    RBT5_STANDARD_WELD_DATA : WORD ;
    RBT6_STANDARD_WELD_DATA : WORD ;
    RBT7_STANDARD_WELD_DATA : WORD ;
    RBT8_STANDARD_WELD_DATA : WORD ;
    RBT9_STANDARD_WELD_DATA : WORD ;
    RBT10_STANDARD_WELD_DATA : WORD ;
    RBT11_STANDARD_WELD_DATA : WORD ;
    RBT12_STANDARD_WELD_DATA : WORD ;
    RBT13_STANDARD_WELD_DATA : WORD ;
    RBT14_STANDARD_WELD_DATA : WORD ;
    RBT15_STANDARD_WELD_DATA : WORD ;
    RBT16_STANDARD_WELD_DATA : WORD ;
    RBT17_STANDARD_WELD_DATA : WORD ;
    RBT18_STANDARD_WELD_DATA : WORD ;
    RBT19_STANDARD_WELD_DATA : WORD ;
    RBT20_STANDARD_WELD_DATA : WORD ;
    RBT21_STANDARD_WELD_DATA : WORD ;
    RBT22_STANDARD_WELD_DATA : WORD ;
    RBT23_STANDARD_WELD_DAT : WORD ;
    RBT24_STANDARD_WELD_DAT : WORD ;
    CHK_WORD : WORD ;
    TEST_TEMP : ARRAY  [1 .. 40 ] OF BYTE ;
   END_STRUCT ;
   S705_BT_CODE_2117 : STRUCT
    STATION_MAIN : WORD ;
    DISTINCTION_LH_RH : WORD ;
    STAION_NUMBER : WORD ;
    BODY_TYPE_1ST : WORD ;
    BODY_TYPE_OPTION : WORD ;
    RBT1_STANDARD_WELD_DATA : WORD ;
    RBT2_STANDARD_WELD_DATA : WORD ;
    RBT3_STANDARD_WELD_DATA : WORD ;
    RBT4_STANDARD_WELD_DATA : WORD ;
    RBT5_STANDARD_WELD_DATA : WORD ;
    RBT6_STANDARD_WELD_DATA : WORD ;
    RBT7_STANDARD_WELD_DATA : WORD ;
    RBT8_STANDARD_WELD_DATA : WORD ;
    RBT9_STANDARD_WELD_DATA : WORD ;
    RBT10_STANDARD_WELD_DATA : WORD ;
    RBT11_STANDARD_WELD_DATA : WORD ;
    RBT12_STANDARD_WELD_DATA : WORD ;
    RBT13_STANDARD_WELD_DATA : WORD ;
    RBT14_STANDARD_WELD_DATA : WORD ;
    RBT15_STANDARD_WELD_DATA : WORD ;
    RBT16_STANDARD_WELD_DATA : WORD ;
    RBT17_STANDARD_WELD_DATA : WORD ;
    RBT18_STANDARD_WELD_DATA : WORD ;
    RBT19_STANDARD_WELD_DATA : WORD ;
    RBT20_STANDARD_WELD_DATA : WORD ;
    RBT21_STANDARD_WELD_DATA : WORD ;
    RBT22_STANDARD_WELD_DATA : WORD ;
    RBT23_STANDARD_WELD_DAT : WORD ;
    RBT24_STANDARD_WELD_DAT : WORD ;
    CHK_WORD : WORD ;
    TEST_TEMP : ARRAY  [1 .. 40 ] OF BYTE ;
   END_STRUCT ;
   S705_BT_CODE_2118 : STRUCT
    STATION_MAIN : WORD ;
    DISTINCTION_LH_RH : WORD ;
    STAION_NUMBER : WORD ;
    BODY_TYPE_1ST : WORD ;
    BODY_TYPE_OPTION : WORD ;
    RBT1_STANDARD_WELD_DATA : WORD ;
    RBT2_STANDARD_WELD_DATA : WORD ;
    RBT3_STANDARD_WELD_DATA : WORD ;
    RBT4_STANDARD_WELD_DATA : WORD ;
    RBT5_STANDARD_WELD_DATA : WORD ;
    RBT6_STANDARD_WELD_DATA : WORD ;
    RBT7_STANDARD_WELD_DATA : WORD ;
    RBT8_STANDARD_WELD_DATA : WORD ;
    RBT9_STANDARD_WELD_DATA : WORD ;
    RBT10_STANDARD_WELD_DATA : WORD ;
    RBT11_STANDARD_WELD_DATA : WORD ;
    RBT12_STANDARD_WELD_DATA : WORD ;
    RBT13_STANDARD_WELD_DATA : WORD ;
    RBT14_STANDARD_WELD_DATA : WORD ;
    RBT15_STANDARD_WELD_DATA : WORD ;
    RBT16_STANDARD_WELD_DATA : WORD ;
    RBT17_STANDARD_WELD_DATA : WORD ;
    RBT18_STANDARD_WELD_DATA : WORD ;
    RBT19_STANDARD_WELD_DATA : WORD ;
    RBT20_STANDARD_WELD_DATA : WORD ;
    RBT21_STANDARD_WELD_DATA : WORD ;
    RBT22_STANDARD_WELD_DATA : WORD ;
    RBT23_STANDARD_WELD_DAT : WORD ;
    RBT24_STANDARD_WELD_DAT : WORD ;
    CHK_WORD : WORD ;
    TEST_TEMP : ARRAY  [1 .. 40 ] OF BYTE ;
   END_STRUCT ;
   S705_BT_CODE_2119 : STRUCT
    STATION_MAIN : WORD ;
    DISTINCTION_LH_RH : WORD ;
    STAION_NUMBER : WORD ;
    BODY_TYPE_1ST : WORD ;
    BODY_TYPE_OPTION : WORD ;
    RBT1_STANDARD_WELD_DATA : WORD ;
    RBT2_STANDARD_WELD_DATA : WORD ;
    RBT3_STANDARD_WELD_DATA : WORD ;
    RBT4_STANDARD_WELD_DATA : WORD ;
    RBT5_STANDARD_WELD_DATA : WORD ;
    RBT6_STANDARD_WELD_DATA : WORD ;
    RBT7_STANDARD_WELD_DATA : WORD ;
    RBT8_STANDARD_WELD_DATA : WORD ;
    RBT9_STANDARD_WELD_DATA : WORD ;
    RBT10_STANDARD_WELD_DATA : WORD ;
    RBT11_STANDARD_WELD_DATA : WORD ;
    RBT12_STANDARD_WELD_DATA : WORD ;
    RBT13_STANDARD_WELD_DATA : WORD ;
    RBT14_STANDARD_WELD_DATA : WORD ;
    RBT15_STANDARD_WELD_DATA : WORD ;
    RBT16_STANDARD_WELD_DATA : WORD ;
    RBT17_STANDARD_WELD_DATA : WORD ;
    RBT18_STANDARD_WELD_DATA : WORD ;
    RBT19_STANDARD_WELD_DATA : WORD ;
    RBT20_STANDARD_WELD_DATA : WORD ;
    RBT21_STANDARD_WELD_DATA : WORD ;
    RBT22_STANDARD_WELD_DATA : WORD ;
    RBT23_STANDARD_WELD_DAT : WORD ;
    RBT24_STANDARD_WELD_DAT : WORD ;
    CHK_WORD : WORD ;
    TEST_TEMP : ARRAY  [1 .. 40 ] OF BYTE ;
   END_STRUCT ;
   S705_BT_CODE_2120 : STRUCT
    STATION_MAIN : WORD ;
    DISTINCTION_LH_RH : WORD ;
    STAION_NUMBER : WORD ;
    BODY_TYPE_1ST : WORD ;
    BODY_TYPE_OPTION : WORD ;
    RBT1_STANDARD_WELD_DATA : WORD ;
    RBT2_STANDARD_WELD_DATA : WORD ;
    RBT3_STANDARD_WELD_DATA : WORD ;
    RBT4_STANDARD_WELD_DATA : WORD ;
    RBT5_STANDARD_WELD_DATA : WORD ;
    RBT6_STANDARD_WELD_DATA : WORD ;
    RBT7_STANDARD_WELD_DATA : WORD ;
    RBT8_STANDARD_WELD_DATA : WORD ;
    RBT9_STANDARD_WELD_DATA : WORD ;
    RBT10_STANDARD_WELD_DATA : WORD ;
    RBT11_STANDARD_WELD_DATA : WORD ;
    RBT12_STANDARD_WELD_DATA : WORD ;
    RBT13_STANDARD_WELD_DATA : WORD ;
    RBT14_STANDARD_WELD_DATA : WORD ;
    RBT15_STANDARD_WELD_DATA : WORD ;
    RBT16_STANDARD_WELD_DATA : WORD ;
    RBT17_STANDARD_WELD_DATA : WORD ;
    RBT18_STANDARD_WELD_DATA : WORD ;
    RBT19_STANDARD_WELD_DATA : WORD ;
    RBT20_STANDARD_WELD_DATA : WORD ;
    RBT21_STANDARD_WELD_DATA : WORD ;
    RBT22_STANDARD_WELD_DATA : WORD ;
    RBT23_STANDARD_WELD_DAT : WORD ;
    RBT24_STANDARD_WELD_DAT : WORD ;
    CHK_WORD : WORD ;
    TEST_TEMP : ARRAY  [1 .. 40 ] OF BYTE ;
   END_STRUCT ;
   S706_BT_CODE_2101 : STRUCT
    STATION_MAIN : WORD ;
    DISTINCTION_LH_RH : WORD ;
    STAION_NUMBER : WORD ;
    BODY_TYPE_1ST : WORD ;
    BODY_TYPE_OPTION : WORD ;
    RBT1_STANDARD_WELD_DATA : WORD ;
    RBT2_STANDARD_WELD_DATA : WORD ;
    RBT3_STANDARD_WELD_DATA : WORD ;
    RBT4_STANDARD_WELD_DATA : WORD ;
    RBT5_STANDARD_WELD_DATA : WORD ;
    RBT6_STANDARD_WELD_DATA : WORD ;
    RBT7_STANDARD_WELD_DATA : WORD ;
    RBT8_STANDARD_WELD_DATA : WORD ;
    RBT9_STANDARD_WELD_DATA : WORD ;
    RBT10_STANDARD_WELD_DATA : WORD ;
    RBT11_STANDARD_WELD_DATA : WORD ;
    RBT12_STANDARD_WELD_DATA : WORD ;
    RBT13_STANDARD_WELD_DATA : WORD ;
    RBT14_STANDARD_WELD_DATA : WORD ;
    RBT15_STANDARD_WELD_DATA : WORD ;
    RBT16_STANDARD_WELD_DATA : WORD ;
    RBT17_STANDARD_WELD_DATA : WORD ;
    RBT18_STANDARD_WELD_DATA : WORD ;
    RBT19_STANDARD_WELD_DATA : WORD ;
    RBT20_STANDARD_WELD_DATA : WORD ;
    RBT21_STANDARD_WELD_DATA : WORD ;
    RBT22_STANDARD_WELD_DATA : WORD ;
    RBT23_STANDARD_WELD_DAT : WORD ;
    RBT24_STANDARD_WELD_DAT : WORD ;
    CHK_WORD : WORD ;
    TEST_TEMP : ARRAY  [1 .. 40 ] OF BYTE ;
   END_STRUCT ;
   S706_BT_CODE_2102 : STRUCT
    STATION_MAIN : WORD ;
    DISTINCTION_LH_RH : WORD ;
    STAION_NUMBER : WORD ;
    BODY_TYPE_1ST : WORD ;
    BODY_TYPE_OPTION : WORD ;
    RBT1_STANDARD_WELD_DATA : WORD ;
    RBT2_STANDARD_WELD_DATA : WORD ;
    RBT3_STANDARD_WELD_DATA : WORD ;
    RBT4_STANDARD_WELD_DATA : WORD ;
    RBT5_STANDARD_WELD_DATA : WORD ;
    RBT6_STANDARD_WELD_DATA : WORD ;
    RBT7_STANDARD_WELD_DATA : WORD ;
    RBT8_STANDARD_WELD_DATA : WORD ;
    RBT9_STANDARD_WELD_DATA : WORD ;
    RBT10_STANDARD_WELD_DATA : WORD ;
    RBT11_STANDARD_WELD_DATA : WORD ;
    RBT12_STANDARD_WELD_DATA : WORD ;
    RBT13_STANDARD_WELD_DATA : WORD ;
    RBT14_STANDARD_WELD_DATA : WORD ;
    RBT15_STANDARD_WELD_DATA : WORD ;
    RBT16_STANDARD_WELD_DATA : WORD ;
    RBT17_STANDARD_WELD_DATA : WORD ;
    RBT18_STANDARD_WELD_DATA : WORD ;
    RBT19_STANDARD_WELD_DATA : WORD ;
    RBT20_STANDARD_WELD_DATA : WORD ;
    RBT21_STANDARD_WELD_DATA : WORD ;
    RBT22_STANDARD_WELD_DATA : WORD ;
    RBT23_STANDARD_WELD_DAT : WORD ;
    RBT24_STANDARD_WELD_DAT : WORD ;
    CHK_WORD : WORD ;
    TEST_TEMP : ARRAY  [1 .. 40 ] OF BYTE ;
   END_STRUCT ;
   S706_BT_CODE_2103 : STRUCT
    STATION_MAIN : WORD ;
    DISTINCTION_LH_RH : WORD ;
    STAION_NUMBER : WORD ;
    BODY_TYPE_1ST : WORD ;
    BODY_TYPE_OPTION : WORD ;
    RBT1_STANDARD_WELD_DATA : WORD ;
    RBT2_STANDARD_WELD_DATA : WORD ;
    RBT3_STANDARD_WELD_DATA : WORD ;
    RBT4_STANDARD_WELD_DATA : WORD ;
    RBT5_STANDARD_WELD_DATA : WORD ;
    RBT6_STANDARD_WELD_DATA : WORD ;
    RBT7_STANDARD_WELD_DATA : WORD ;
    RBT8_STANDARD_WELD_DATA : WORD ;
    RBT9_STANDARD_WELD_DATA : WORD ;
    RBT10_STANDARD_WELD_DATA : WORD ;
    RBT11_STANDARD_WELD_DATA : WORD ;
    RBT12_STANDARD_WELD_DATA : WORD ;
    RBT13_STANDARD_WELD_DATA : WORD ;
    RBT14_STANDARD_WELD_DATA : WORD ;
    RBT15_STANDARD_WELD_DATA : WORD ;
    RBT16_STANDARD_WELD_DATA : WORD ;
    RBT17_STANDARD_WELD_DATA : WORD ;
    RBT18_STANDARD_WELD_DATA : WORD ;
    RBT19_STANDARD_WELD_DATA : WORD ;
    RBT20_STANDARD_WELD_DATA : WORD ;
    RBT21_STANDARD_WELD_DATA : WORD ;
    RBT22_STANDARD_WELD_DATA : WORD ;
    RBT23_STANDARD_WELD_DAT : WORD ;
    RBT24_STANDARD_WELD_DAT : WORD ;
    CHK_WORD : WORD ;
    TEST_TEMP : ARRAY  [1 .. 40 ] OF BYTE ;
   END_STRUCT ;
   S706_BT_CODE_2104 : STRUCT
    STATION_MAIN : WORD ;
    DISTINCTION_LH_RH : WORD ;
    STAION_NUMBER : WORD ;
    BODY_TYPE_1ST : WORD ;
    BODY_TYPE_OPTION : WORD ;
    RBT1_STANDARD_WELD_DATA : WORD ;
    RBT2_STANDARD_WELD_DATA : WORD ;
    RBT3_STANDARD_WELD_DATA : WORD ;
    RBT4_STANDARD_WELD_DATA : WORD ;
    RBT5_STANDARD_WELD_DATA : WORD ;
    RBT6_STANDARD_WELD_DATA : WORD ;
    RBT7_STANDARD_WELD_DATA : WORD ;
    RBT8_STANDARD_WELD_DATA : WORD ;
    RBT9_STANDARD_WELD_DATA : WORD ;
    RBT10_STANDARD_WELD_DATA : WORD ;
    RBT11_STANDARD_WELD_DATA : WORD ;
    RBT12_STANDARD_WELD_DATA : WORD ;
    RBT13_STANDARD_WELD_DATA : WORD ;
    RBT14_STANDARD_WELD_DATA : WORD ;
    RBT15_STANDARD_WELD_DATA : WORD ;
    RBT16_STANDARD_WELD_DATA : WORD ;
    RBT17_STANDARD_WELD_DATA : WORD ;
    RBT18_STANDARD_WELD_DATA : WORD ;
    RBT19_STANDARD_WELD_DATA : WORD ;
    RBT20_STANDARD_WELD_DATA : WORD ;
    RBT21_STANDARD_WELD_DATA : WORD ;
    RBT22_STANDARD_WELD_DATA : WORD ;
    RBT23_STANDARD_WELD_DAT : WORD ;
    RBT24_STANDARD_WELD_DAT : WORD ;
    CHK_WORD : WORD ;
    TEST_TEMP : ARRAY  [1 .. 40 ] OF BYTE ;
   END_STRUCT ;
   S706_BT_CODE_2105 : STRUCT
    STATION_MAIN : WORD ;
    DISTINCTION_LH_RH : WORD ;
    STAION_NUMBER : WORD ;
    BODY_TYPE_1ST : WORD ;
    BODY_TYPE_OPTION : WORD ;
    RBT1_STANDARD_WELD_DATA : WORD ;
    RBT2_STANDARD_WELD_DATA : WORD ;
    RBT3_STANDARD_WELD_DATA : WORD ;
    RBT4_STANDARD_WELD_DATA : WORD ;
    RBT5_STANDARD_WELD_DATA : WORD ;
    RBT6_STANDARD_WELD_DATA : WORD ;
    RBT7_STANDARD_WELD_DATA : WORD ;
    RBT8_STANDARD_WELD_DATA : WORD ;
    RBT9_STANDARD_WELD_DATA : WORD ;
    RBT10_STANDARD_WELD_DATA : WORD ;
    RBT11_STANDARD_WELD_DATA : WORD ;
    RBT12_STANDARD_WELD_DATA : WORD ;
    RBT13_STANDARD_WELD_DATA : WORD ;
    RBT14_STANDARD_WELD_DATA : WORD ;
    RBT15_STANDARD_WELD_DATA : WORD ;
    RBT16_STANDARD_WELD_DATA : WORD ;
    RBT17_STANDARD_WELD_DATA : WORD ;
    RBT18_STANDARD_WELD_DATA : WORD ;
    RBT19_STANDARD_WELD_DATA : WORD ;
    RBT20_STANDARD_WELD_DATA : WORD ;
    RBT21_STANDARD_WELD_DATA : WORD ;
    RBT22_STANDARD_WELD_DATA : WORD ;
    RBT23_STANDARD_WELD_DAT : WORD ;
    RBT24_STANDARD_WELD_DAT : WORD ;
    CHK_WORD : WORD ;
    TEST_TEMP : ARRAY  [1 .. 40 ] OF BYTE ;
   END_STRUCT ;
   S706_BT_CODE_2106 : STRUCT
    STATION_MAIN : WORD ;
    DISTINCTION_LH_RH : WORD ;
    STAION_NUMBER : WORD ;
    BODY_TYPE_1ST : WORD ;
    BODY_TYPE_OPTION : WORD ;
    RBT1_STANDARD_WELD_DATA : WORD ;
    RBT2_STANDARD_WELD_DATA : WORD ;
    RBT3_STANDARD_WELD_DATA : WORD ;
    RBT4_STANDARD_WELD_DATA : WORD ;
    RBT5_STANDARD_WELD_DATA : WORD ;
    RBT6_STANDARD_WELD_DATA : WORD ;
    RBT7_STANDARD_WELD_DATA : WORD ;
    RBT8_STANDARD_WELD_DATA : WORD ;
    RBT9_STANDARD_WELD_DATA : WORD ;
    RBT10_STANDARD_WELD_DATA : WORD ;
    RBT11_STANDARD_WELD_DATA : WORD ;
    RBT12_STANDARD_WELD_DATA : WORD ;
    RBT13_STANDARD_WELD_DATA : WORD ;
    RBT14_STANDARD_WELD_DATA : WORD ;
    RBT15_STANDARD_WELD_DATA : WORD ;
    RBT16_STANDARD_WELD_DATA : WORD ;
    RBT17_STANDARD_WELD_DATA : WORD ;
    RBT18_STANDARD_WELD_DATA : WORD ;
    RBT19_STANDARD_WELD_DATA : WORD ;
    RBT20_STANDARD_WELD_DATA : WORD ;
    RBT21_STANDARD_WELD_DATA : WORD ;
    RBT22_STANDARD_WELD_DATA : WORD ;
    RBT23_STANDARD_WELD_DAT : WORD ;
    RBT24_STANDARD_WELD_DAT : WORD ;
    CHK_WORD : WORD ;
    TEST_TEMP : ARRAY  [1 .. 40 ] OF BYTE ;
   END_STRUCT ;
   S706_BT_CODE_2107 : STRUCT
    STATION_MAIN : WORD ;
    DISTINCTION_LH_RH : WORD ;
    STAION_NUMBER : WORD ;
    BODY_TYPE_1ST : WORD ;
    BODY_TYPE_OPTION : WORD ;
    RBT1_STANDARD_WELD_DATA : WORD ;
    RBT2_STANDARD_WELD_DATA : WORD ;
    RBT3_STANDARD_WELD_DATA : WORD ;
    RBT4_STANDARD_WELD_DATA : WORD ;
    RBT5_STANDARD_WELD_DATA : WORD ;
    RBT6_STANDARD_WELD_DATA : WORD ;
    RBT7_STANDARD_WELD_DATA : WORD ;
    RBT8_STANDARD_WELD_DATA : WORD ;
    RBT9_STANDARD_WELD_DATA : WORD ;
    RBT10_STANDARD_WELD_DATA : WORD ;
    RBT11_STANDARD_WELD_DATA : WORD ;
    RBT12_STANDARD_WELD_DATA : WORD ;
    RBT13_STANDARD_WELD_DATA : WORD ;
    RBT14_STANDARD_WELD_DATA : WORD ;
    RBT15_STANDARD_WELD_DATA : WORD ;
    RBT16_STANDARD_WELD_DATA : WORD ;
    RBT17_STANDARD_WELD_DATA : WORD ;
    RBT18_STANDARD_WELD_DATA : WORD ;
    RBT19_STANDARD_WELD_DATA : WORD ;
    RBT20_STANDARD_WELD_DATA : WORD ;
    RBT21_STANDARD_WELD_DATA : WORD ;
    RBT22_STANDARD_WELD_DATA : WORD ;
    RBT23_STANDARD_WELD_DAT : WORD ;
    RBT24_STANDARD_WELD_DAT : WORD ;
    CHK_WORD : WORD ;
    TEST_TEMP : ARRAY  [1 .. 40 ] OF BYTE ;
   END_STRUCT ;
   S706_BT_CODE_2108 : STRUCT
    STATION_MAIN : WORD ;
    DISTINCTION_LH_RH : WORD ;
    STAION_NUMBER : WORD ;
    BODY_TYPE_1ST : WORD ;
    BODY_TYPE_OPTION : WORD ;
    RBT1_STANDARD_WELD_DATA : WORD ;
    RBT2_STANDARD_WELD_DATA : WORD ;
    RBT3_STANDARD_WELD_DATA : WORD ;
    RBT4_STANDARD_WELD_DATA : WORD ;
    RBT5_STANDARD_WELD_DATA : WORD ;
    RBT6_STANDARD_WELD_DATA : WORD ;
    RBT7_STANDARD_WELD_DATA : WORD ;
    RBT8_STANDARD_WELD_DATA : WORD ;
    RBT9_STANDARD_WELD_DATA : WORD ;
    RBT10_STANDARD_WELD_DATA : WORD ;
    RBT11_STANDARD_WELD_DATA : WORD ;
    RBT12_STANDARD_WELD_DATA : WORD ;
    RBT13_STANDARD_WELD_DATA : WORD ;
    RBT14_STANDARD_WELD_DATA : WORD ;
    RBT15_STANDARD_WELD_DATA : WORD ;
    RBT16_STANDARD_WELD_DATA : WORD ;
    RBT17_STANDARD_WELD_DATA : WORD ;
    RBT18_STANDARD_WELD_DATA : WORD ;
    RBT19_STANDARD_WELD_DATA : WORD ;
    RBT20_STANDARD_WELD_DATA : WORD ;
    RBT21_STANDARD_WELD_DATA : WORD ;
    RBT22_STANDARD_WELD_DATA : WORD ;
    RBT23_STANDARD_WELD_DAT : WORD ;
    RBT24_STANDARD_WELD_DAT : WORD ;
    CHK_WORD : WORD ;
    TEST_TEMP : ARRAY  [1 .. 40 ] OF BYTE ;
   END_STRUCT ;
   S706_BT_CODE_2109 : STRUCT
    STATION_MAIN : WORD ;
    DISTINCTION_LH_RH : WORD ;
    STAION_NUMBER : WORD ;
    BODY_TYPE_1ST : WORD ;
    BODY_TYPE_OPTION : WORD ;
    RBT1_STANDARD_WELD_DATA : WORD ;
    RBT2_STANDARD_WELD_DATA : WORD ;
    RBT3_STANDARD_WELD_DATA : WORD ;
    RBT4_STANDARD_WELD_DATA : WORD ;
    RBT5_STANDARD_WELD_DATA : WORD ;
    RBT6_STANDARD_WELD_DATA : WORD ;
    RBT7_STANDARD_WELD_DATA : WORD ;
    RBT8_STANDARD_WELD_DATA : WORD ;
    RBT9_STANDARD_WELD_DATA : WORD ;
    RBT10_STANDARD_WELD_DATA : WORD ;
    RBT11_STANDARD_WELD_DATA : WORD ;
    RBT12_STANDARD_WELD_DATA : WORD ;
    RBT13_STANDARD_WELD_DATA : WORD ;
    RBT14_STANDARD_WELD_DATA : WORD ;
    RBT15_STANDARD_WELD_DATA : WORD ;
    RBT16_STANDARD_WELD_DATA : WORD ;
    RBT17_STANDARD_WELD_DATA : WORD ;
    RBT18_STANDARD_WELD_DATA : WORD ;
    RBT19_STANDARD_WELD_DATA : WORD ;
    RBT20_STANDARD_WELD_DATA : WORD ;
    RBT21_STANDARD_WELD_DATA : WORD ;
    RBT22_STANDARD_WELD_DATA : WORD ;
    RBT23_STANDARD_WELD_DAT : WORD ;
    RBT24_STANDARD_WELD_DAT : WORD ;
    CHK_WORD : WORD ;
    TEST_TEMP : ARRAY  [1 .. 40 ] OF BYTE ;
   END_STRUCT ;
   S706_BT_CODE_2110 : STRUCT
    STATION_MAIN : WORD ;
    DISTINCTION_LH_RH : WORD ;
    STAION_NUMBER : WORD ;
    BODY_TYPE_1ST : WORD ;
    BODY_TYPE_OPTION : WORD ;
    RBT1_STANDARD_WELD_DATA : WORD ;
    RBT2_STANDARD_WELD_DATA : WORD ;
    RBT3_STANDARD_WELD_DATA : WORD ;
    RBT4_STANDARD_WELD_DATA : WORD ;
    RBT5_STANDARD_WELD_DATA : WORD ;
    RBT6_STANDARD_WELD_DATA : WORD ;
    RBT7_STANDARD_WELD_DATA : WORD ;
    RBT8_STANDARD_WELD_DATA : WORD ;
    RBT9_STANDARD_WELD_DATA : WORD ;
    RBT10_STANDARD_WELD_DATA : WORD ;
    RBT11_STANDARD_WELD_DATA : WORD ;
    RBT12_STANDARD_WELD_DATA : WORD ;
    RBT13_STANDARD_WELD_DATA : WORD ;
    RBT14_STANDARD_WELD_DATA : WORD ;
    RBT15_STANDARD_WELD_DATA : WORD ;
    RBT16_STANDARD_WELD_DATA : WORD ;
    RBT17_STANDARD_WELD_DATA : WORD ;
    RBT18_STANDARD_WELD_DATA : WORD ;
    RBT19_STANDARD_WELD_DATA : WORD ;
    RBT20_STANDARD_WELD_DATA : WORD ;
    RBT21_STANDARD_WELD_DATA : WORD ;
    RBT22_STANDARD_WELD_DATA : WORD ;
    RBT23_STANDARD_WELD_DAT : WORD ;
    RBT24_STANDARD_WELD_DAT : WORD ;
    CHK_WORD : WORD ;
    TEST_TEMP : ARRAY  [1 .. 40 ] OF BYTE ;
   END_STRUCT ;
   S706_BT_CODE_2111 : STRUCT
    STATION_MAIN : WORD ;
    DISTINCTION_LH_RH : WORD ;
    STAION_NUMBER : WORD ;
    BODY_TYPE_1ST : WORD ;
    BODY_TYPE_OPTION : WORD ;
    RBT1_STANDARD_WELD_DATA : WORD ;
    RBT2_STANDARD_WELD_DATA : WORD ;
    RBT3_STANDARD_WELD_DATA : WORD ;
    RBT4_STANDARD_WELD_DATA : WORD ;
    RBT5_STANDARD_WELD_DATA : WORD ;
    RBT6_STANDARD_WELD_DATA : WORD ;
    RBT7_STANDARD_WELD_DATA : WORD ;
    RBT8_STANDARD_WELD_DATA : WORD ;
    RBT9_STANDARD_WELD_DATA : WORD ;
    RBT10_STANDARD_WELD_DATA : WORD ;
    RBT11_STANDARD_WELD_DATA : WORD ;
    RBT12_STANDARD_WELD_DATA : WORD ;
    RBT13_STANDARD_WELD_DATA : WORD ;
    RBT14_STANDARD_WELD_DATA : WORD ;
    RBT15_STANDARD_WELD_DATA : WORD ;
    RBT16_STANDARD_WELD_DATA : WORD ;
    RBT17_STANDARD_WELD_DATA : WORD ;
    RBT18_STANDARD_WELD_DATA : WORD ;
    RBT19_STANDARD_WELD_DATA : WORD ;
    RBT20_STANDARD_WELD_DATA : WORD ;
    RBT21_STANDARD_WELD_DATA : WORD ;
    RBT22_STANDARD_WELD_DATA : WORD ;
    RBT23_STANDARD_WELD_DAT : WORD ;
    RBT24_STANDARD_WELD_DAT : WORD ;
    CHK_WORD : WORD ;
    TEST_TEMP : ARRAY  [1 .. 40 ] OF BYTE ;
   END_STRUCT ;
   S706_BT_CODE_2112 : STRUCT
    STATION_MAIN : WORD ;
    DISTINCTION_LH_RH : WORD ;
    STAION_NUMBER : WORD ;
    BODY_TYPE_1ST : WORD ;
    BODY_TYPE_OPTION : WORD ;
    RBT1_STANDARD_WELD_DATA : WORD ;
    RBT2_STANDARD_WELD_DATA : WORD ;
    RBT3_STANDARD_WELD_DATA : WORD ;
    RBT4_STANDARD_WELD_DATA : WORD ;
    RBT5_STANDARD_WELD_DATA : WORD ;
    RBT6_STANDARD_WELD_DATA : WORD ;
    RBT7_STANDARD_WELD_DATA : WORD ;
    RBT8_STANDARD_WELD_DATA : WORD ;
    RBT9_STANDARD_WELD_DATA : WORD ;
    RBT10_STANDARD_WELD_DATA : WORD ;
    RBT11_STANDARD_WELD_DATA : WORD ;
    RBT12_STANDARD_WELD_DATA : WORD ;
    RBT13_STANDARD_WELD_DATA : WORD ;
    RBT14_STANDARD_WELD_DATA : WORD ;
    RBT15_STANDARD_WELD_DATA : WORD ;
    RBT16_STANDARD_WELD_DATA : WORD ;
    RBT17_STANDARD_WELD_DATA : WORD ;
    RBT18_STANDARD_WELD_DATA : WORD ;
    RBT19_STANDARD_WELD_DATA : WORD ;
    RBT20_STANDARD_WELD_DATA : WORD ;
    RBT21_STANDARD_WELD_DATA : WORD ;
    RBT22_STANDARD_WELD_DATA : WORD ;
    RBT23_STANDARD_WELD_DAT : WORD ;
    RBT24_STANDARD_WELD_DAT : WORD ;
    CHK_WORD : WORD ;
    TEST_TEMP : ARRAY  [1 .. 40 ] OF BYTE ;
   END_STRUCT ;
   S706_BT_CODE_2113 : STRUCT
    STATION_MAIN : WORD ;
    DISTINCTION_LH_RH : WORD ;
    STAION_NUMBER : WORD ;
    BODY_TYPE_1ST : WORD ;
    BODY_TYPE_OPTION : WORD ;
    RBT1_STANDARD_WELD_DATA : WORD ;
    RBT2_STANDARD_WELD_DATA : WORD ;
    RBT3_STANDARD_WELD_DATA : WORD ;
    RBT4_STANDARD_WELD_DATA : WORD ;
    RBT5_STANDARD_WELD_DATA : WORD ;
    RBT6_STANDARD_WELD_DATA : WORD ;
    RBT7_STANDARD_WELD_DATA : WORD ;
    RBT8_STANDARD_WELD_DATA : WORD ;
    RBT9_STANDARD_WELD_DATA : WORD ;
    RBT10_STANDARD_WELD_DATA : WORD ;
    RBT11_STANDARD_WELD_DATA : WORD ;
    RBT12_STANDARD_WELD_DATA : WORD ;
    RBT13_STANDARD_WELD_DATA : WORD ;
    RBT14_STANDARD_WELD_DATA : WORD ;
    RBT15_STANDARD_WELD_DATA : WORD ;
    RBT16_STANDARD_WELD_DATA : WORD ;
    RBT17_STANDARD_WELD_DATA : WORD ;
    RBT18_STANDARD_WELD_DATA : WORD ;
    RBT19_STANDARD_WELD_DATA : WORD ;
    RBT20_STANDARD_WELD_DATA : WORD ;
    RBT21_STANDARD_WELD_DATA : WORD ;
    RBT22_STANDARD_WELD_DATA : WORD ;
    RBT23_STANDARD_WELD_DAT : WORD ;
    RBT24_STANDARD_WELD_DAT : WORD ;
    CHK_WORD : WORD ;
    TEST_TEMP : ARRAY  [1 .. 40 ] OF BYTE ;
   END_STRUCT ;
   S706_BT_CODE_2114 : STRUCT
    STATION_MAIN : WORD ;
    DISTINCTION_LH_RH : WORD ;
    STAION_NUMBER : WORD ;
    BODY_TYPE_1ST : WORD ;
    BODY_TYPE_OPTION : WORD ;
    RBT1_STANDARD_WELD_DATA : WORD ;
    RBT2_STANDARD_WELD_DATA : WORD ;
    RBT3_STANDARD_WELD_DATA : WORD ;
    RBT4_STANDARD_WELD_DATA : WORD ;
    RBT5_STANDARD_WELD_DATA : WORD ;
    RBT6_STANDARD_WELD_DATA : WORD ;
    RBT7_STANDARD_WELD_DATA : WORD ;
    RBT8_STANDARD_WELD_DATA : WORD ;
    RBT9_STANDARD_WELD_DATA : WORD ;
    RBT10_STANDARD_WELD_DATA : WORD ;
    RBT11_STANDARD_WELD_DATA : WORD ;
    RBT12_STANDARD_WELD_DATA : WORD ;
    RBT13_STANDARD_WELD_DATA : WORD ;
    RBT14_STANDARD_WELD_DATA : WORD ;
    RBT15_STANDARD_WELD_DATA : WORD ;
    RBT16_STANDARD_WELD_DATA : WORD ;
    RBT17_STANDARD_WELD_DATA : WORD ;
    RBT18_STANDARD_WELD_DATA : WORD ;
    RBT19_STANDARD_WELD_DATA : WORD ;
    RBT20_STANDARD_WELD_DATA : WORD ;
    RBT21_STANDARD_WELD_DATA : WORD ;
    RBT22_STANDARD_WELD_DATA : WORD ;
    RBT23_STANDARD_WELD_DAT : WORD ;
    RBT24_STANDARD_WELD_DAT : WORD ;
    CHK_WORD : WORD ;
    TEST_TEMP : ARRAY  [1 .. 40 ] OF BYTE ;
   END_STRUCT ;
   S706_BT_CODE_2115 : STRUCT
    STATION_MAIN : WORD ;
    DISTINCTION_LH_RH : WORD ;
    STAION_NUMBER : WORD ;
    BODY_TYPE_1ST : WORD ;
    BODY_TYPE_OPTION : WORD ;
    RBT1_STANDARD_WELD_DATA : WORD ;
    RBT2_STANDARD_WELD_DATA : WORD ;
    RBT3_STANDARD_WELD_DATA : WORD ;
    RBT4_STANDARD_WELD_DATA : WORD ;
    RBT5_STANDARD_WELD_DATA : WORD ;
    RBT6_STANDARD_WELD_DATA : WORD ;
    RBT7_STANDARD_WELD_DATA : WORD ;
    RBT8_STANDARD_WELD_DATA : WORD ;
    RBT9_STANDARD_WELD_DATA : WORD ;
    RBT10_STANDARD_WELD_DATA : WORD ;
    RBT11_STANDARD_WELD_DATA : WORD ;
    RBT12_STANDARD_WELD_DATA : WORD ;
    RBT13_STANDARD_WELD_DATA : WORD ;
    RBT14_STANDARD_WELD_DATA : WORD ;
    RBT15_STANDARD_WELD_DATA : WORD ;
    RBT16_STANDARD_WELD_DATA : WORD ;
    RBT17_STANDARD_WELD_DATA : WORD ;
    RBT18_STANDARD_WELD_DATA : WORD ;
    RBT19_STANDARD_WELD_DATA : WORD ;
    RBT20_STANDARD_WELD_DATA : WORD ;
    RBT21_STANDARD_WELD_DATA : WORD ;
    RBT22_STANDARD_WELD_DATA : WORD ;
    RBT23_STANDARD_WELD_DAT : WORD ;
    RBT24_STANDARD_WELD_DAT : WORD ;
    CHK_WORD : WORD ;
    TEST_TEMP : ARRAY  [1 .. 40 ] OF BYTE ;
   END_STRUCT ;
   S706_BT_CODE_2116 : STRUCT
    STATION_MAIN : WORD ;
    DISTINCTION_LH_RH : WORD ;
    STAION_NUMBER : WORD ;
    BODY_TYPE_1ST : WORD ;
    BODY_TYPE_OPTION : WORD ;
    RBT1_STANDARD_WELD_DATA : WORD ;
    RBT2_STANDARD_WELD_DATA : WORD ;
    RBT3_STANDARD_WELD_DATA : WORD ;
    RBT4_STANDARD_WELD_DATA : WORD ;
    RBT5_STANDARD_WELD_DATA : WORD ;
    RBT6_STANDARD_WELD_DATA : WORD ;
    RBT7_STANDARD_WELD_DATA : WORD ;
    RBT8_STANDARD_WELD_DATA : WORD ;
    RBT9_STANDARD_WELD_DATA : WORD ;
    RBT10_STANDARD_WELD_DATA : WORD ;
    RBT11_STANDARD_WELD_DATA : WORD ;
    RBT12_STANDARD_WELD_DATA : WORD ;
    RBT13_STANDARD_WELD_DATA : WORD ;
    RBT14_STANDARD_WELD_DATA : WORD ;
    RBT15_STANDARD_WELD_DATA : WORD ;
    RBT16_STANDARD_WELD_DATA : WORD ;
    RBT17_STANDARD_WELD_DATA : WORD ;
    RBT18_STANDARD_WELD_DATA : WORD ;
    RBT19_STANDARD_WELD_DATA : WORD ;
    RBT20_STANDARD_WELD_DATA : WORD ;
    RBT21_STANDARD_WELD_DATA : WORD ;
    RBT22_STANDARD_WELD_DATA : WORD ;
    RBT23_STANDARD_WELD_DAT : WORD ;
    RBT24_STANDARD_WELD_DAT : WORD ;
    CHK_WORD : WORD ;
    TEST_TEMP : ARRAY  [1 .. 40 ] OF BYTE ;
   END_STRUCT ;
   S706_BT_CODE_2117 : STRUCT
    STATION_MAIN : WORD ;
    DISTINCTION_LH_RH : WORD ;
    STAION_NUMBER : WORD ;
    BODY_TYPE_1ST : WORD ;
    BODY_TYPE_OPTION : WORD ;
    RBT1_STANDARD_WELD_DATA : WORD ;
    RBT2_STANDARD_WELD_DATA : WORD ;
    RBT3_STANDARD_WELD_DATA : WORD ;
    RBT4_STANDARD_WELD_DATA : WORD ;
    RBT5_STANDARD_WELD_DATA : WORD ;
    RBT6_STANDARD_WELD_DATA : WORD ;
    RBT7_STANDARD_WELD_DATA : WORD ;
    RBT8_STANDARD_WELD_DATA : WORD ;
    RBT9_STANDARD_WELD_DATA : WORD ;
    RBT10_STANDARD_WELD_DATA : WORD ;
    RBT11_STANDARD_WELD_DATA : WORD ;
    RBT12_STANDARD_WELD_DATA : WORD ;
    RBT13_STANDARD_WELD_DATA : WORD ;
    RBT14_STANDARD_WELD_DATA : WORD ;
    RBT15_STANDARD_WELD_DATA : WORD ;
    RBT16_STANDARD_WELD_DATA : WORD ;
    RBT17_STANDARD_WELD_DATA : WORD ;
    RBT18_STANDARD_WELD_DATA : WORD ;
    RBT19_STANDARD_WELD_DATA : WORD ;
    RBT20_STANDARD_WELD_DATA : WORD ;
    RBT21_STANDARD_WELD_DATA : WORD ;
    RBT22_STANDARD_WELD_DATA : WORD ;
    RBT23_STANDARD_WELD_DAT : WORD ;
    RBT24_STANDARD_WELD_DAT : WORD ;
    CHK_WORD : WORD ;
    TEST_TEMP : ARRAY  [1 .. 40 ] OF BYTE ;
   END_STRUCT ;
   S706_BT_CODE_2118 : STRUCT
    STATION_MAIN : WORD ;
    DISTINCTION_LH_RH : WORD ;
    STAION_NUMBER : WORD ;
    BODY_TYPE_1ST : WORD ;
    BODY_TYPE_OPTION : WORD ;
    RBT1_STANDARD_WELD_DATA : WORD ;
    RBT2_STANDARD_WELD_DATA : WORD ;
    RBT3_STANDARD_WELD_DATA : WORD ;
    RBT4_STANDARD_WELD_DATA : WORD ;
    RBT5_STANDARD_WELD_DATA : WORD ;
    RBT6_STANDARD_WELD_DATA : WORD ;
    RBT7_STANDARD_WELD_DATA : WORD ;
    RBT8_STANDARD_WELD_DATA : WORD ;
    RBT9_STANDARD_WELD_DATA : WORD ;
    RBT10_STANDARD_WELD_DATA : WORD ;
    RBT11_STANDARD_WELD_DATA : WORD ;
    RBT12_STANDARD_WELD_DATA : WORD ;
    RBT13_STANDARD_WELD_DATA : WORD ;
    RBT14_STANDARD_WELD_DATA : WORD ;
    RBT15_STANDARD_WELD_DATA : WORD ;
    RBT16_STANDARD_WELD_DATA : WORD ;
    RBT17_STANDARD_WELD_DATA : WORD ;
    RBT18_STANDARD_WELD_DATA : WORD ;
    RBT19_STANDARD_WELD_DATA : WORD ;
    RBT20_STANDARD_WELD_DATA : WORD ;
    RBT21_STANDARD_WELD_DATA : WORD ;
    RBT22_STANDARD_WELD_DATA : WORD ;
    RBT23_STANDARD_WELD_DAT : WORD ;
    RBT24_STANDARD_WELD_DAT : WORD ;
    CHK_WORD : WORD ;
    TEST_TEMP : ARRAY  [1 .. 40 ] OF BYTE ;
   END_STRUCT ;
   S706_BT_CODE_2119 : STRUCT
    STATION_MAIN : WORD ;
    DISTINCTION_LH_RH : WORD ;
    STAION_NUMBER : WORD ;
    BODY_TYPE_1ST : WORD ;
    BODY_TYPE_OPTION : WORD ;
    RBT1_STANDARD_WELD_DATA : WORD ;
    RBT2_STANDARD_WELD_DATA : WORD ;
    RBT3_STANDARD_WELD_DATA : WORD ;
    RBT4_STANDARD_WELD_DATA : WORD ;
    RBT5_STANDARD_WELD_DATA : WORD ;
    RBT6_STANDARD_WELD_DATA : WORD ;
    RBT7_STANDARD_WELD_DATA : WORD ;
    RBT8_STANDARD_WELD_DATA : WORD ;
    RBT9_STANDARD_WELD_DATA : WORD ;
    RBT10_STANDARD_WELD_DATA : WORD ;
    RBT11_STANDARD_WELD_DATA : WORD ;
    RBT12_STANDARD_WELD_DATA : WORD ;
    RBT13_STANDARD_WELD_DATA : WORD ;
    RBT14_STANDARD_WELD_DATA : WORD ;
    RBT15_STANDARD_WELD_DATA : WORD ;
    RBT16_STANDARD_WELD_DATA : WORD ;
    RBT17_STANDARD_WELD_DATA : WORD ;
    RBT18_STANDARD_WELD_DATA : WORD ;
    RBT19_STANDARD_WELD_DATA : WORD ;
    RBT20_STANDARD_WELD_DATA : WORD ;
    RBT21_STANDARD_WELD_DATA : WORD ;
    RBT22_STANDARD_WELD_DATA : WORD ;
    RBT23_STANDARD_WELD_DAT : WORD ;
    RBT24_STANDARD_WELD_DAT : WORD ;
    CHK_WORD : WORD ;
    TEST_TEMP : ARRAY  [1 .. 40 ] OF BYTE ;
   END_STRUCT ;
   S706_BT_CODE_2120 : STRUCT
    STATION_MAIN : WORD ;
    DISTINCTION_LH_RH : WORD ;
    STAION_NUMBER : WORD ;
    BODY_TYPE_1ST : WORD ;
    BODY_TYPE_OPTION : WORD ;
    RBT1_STANDARD_WELD_DATA : WORD ;
    RBT2_STANDARD_WELD_DATA : WORD ;
    RBT3_STANDARD_WELD_DATA : WORD ;
    RBT4_STANDARD_WELD_DATA : WORD ;
    RBT5_STANDARD_WELD_DATA : WORD ;
    RBT6_STANDARD_WELD_DATA : WORD ;
    RBT7_STANDARD_WELD_DATA : WORD ;
    RBT8_STANDARD_WELD_DATA : WORD ;
    RBT9_STANDARD_WELD_DATA : WORD ;
    RBT10_STANDARD_WELD_DATA : WORD ;
    RBT11_STANDARD_WELD_DATA : WORD ;
    RBT12_STANDARD_WELD_DATA : WORD ;
    RBT13_STANDARD_WELD_DATA : WORD ;
    RBT14_STANDARD_WELD_DATA : WORD ;
    RBT15_STANDARD_WELD_DATA : WORD ;
    RBT16_STANDARD_WELD_DATA : WORD ;
    RBT17_STANDARD_WELD_DATA : WORD ;
    RBT18_STANDARD_WELD_DATA : WORD ;
    RBT19_STANDARD_WELD_DATA : WORD ;
    RBT20_STANDARD_WELD_DATA : WORD ;
    RBT21_STANDARD_WELD_DATA : WORD ;
    RBT22_STANDARD_WELD_DATA : WORD ;
    RBT23_STANDARD_WELD_DAT : WORD ;
    RBT24_STANDARD_WELD_DAT : WORD ;
    CHK_WORD : WORD ;
    TEST_TEMP : ARRAY  [1 .. 40 ] OF BYTE ;
   END_STRUCT ;
   S707_BT_CODE_2101 : STRUCT
    STATION_MAIN : WORD ;
    DISTINCTION_LH_RH : WORD ;
    STAION_NUMBER : WORD ;
    BODY_TYPE_1ST : WORD ;
    BODY_TYPE_OPTION : WORD ;
    RBT1_STANDARD_WELD_DATA : WORD ;
    RBT2_STANDARD_WELD_DATA : WORD ;
    RBT3_STANDARD_WELD_DATA : WORD ;
    RBT4_STANDARD_WELD_DATA : WORD ;
    RBT5_STANDARD_WELD_DATA : WORD ;
    RBT6_STANDARD_WELD_DATA : WORD ;
    RBT7_STANDARD_WELD_DATA : WORD ;
    RBT8_STANDARD_WELD_DATA : WORD ;
    RBT9_STANDARD_WELD_DATA : WORD ;
    RBT10_STANDARD_WELD_DATA : WORD ;
    RBT11_STANDARD_WELD_DATA : WORD ;
    RBT12_STANDARD_WELD_DATA : WORD ;
    RBT13_STANDARD_WELD_DATA : WORD ;
    RBT14_STANDARD_WELD_DATA : WORD ;
    RBT15_STANDARD_WELD_DATA : WORD ;
    RBT16_STANDARD_WELD_DATA : WORD ;
    RBT17_STANDARD_WELD_DATA : WORD ;
    RBT18_STANDARD_WELD_DATA : WORD ;
    RBT19_STANDARD_WELD_DATA : WORD ;
    RBT20_STANDARD_WELD_DATA : WORD ;
    RBT21_STANDARD_WELD_DATA : WORD ;
    RBT22_STANDARD_WELD_DATA : WORD ;
    RBT23_STANDARD_WELD_DAT : WORD ;
    RBT24_STANDARD_WELD_DAT : WORD ;
    CHK_WORD : WORD ;
    TEST_TEMP : ARRAY  [1 .. 40 ] OF BYTE ;
   END_STRUCT ;
   S707_BT_CODE_2102 : STRUCT
    STATION_MAIN : WORD ;
    DISTINCTION_LH_RH : WORD ;
    STAION_NUMBER : WORD ;
    BODY_TYPE_1ST : WORD ;
    BODY_TYPE_OPTION : WORD ;
    RBT1_STANDARD_WELD_DATA : WORD ;
    RBT2_STANDARD_WELD_DATA : WORD ;
    RBT3_STANDARD_WELD_DATA : WORD ;
    RBT4_STANDARD_WELD_DATA : WORD ;
    RBT5_STANDARD_WELD_DATA : WORD ;
    RBT6_STANDARD_WELD_DATA : WORD ;
    RBT7_STANDARD_WELD_DATA : WORD ;
    RBT8_STANDARD_WELD_DATA : WORD ;
    RBT9_STANDARD_WELD_DATA : WORD ;
    RBT10_STANDARD_WELD_DATA : WORD ;
    RBT11_STANDARD_WELD_DATA : WORD ;
    RBT12_STANDARD_WELD_DATA : WORD ;
    RBT13_STANDARD_WELD_DATA : WORD ;
    RBT14_STANDARD_WELD_DATA : WORD ;
    RBT15_STANDARD_WELD_DATA : WORD ;
    RBT16_STANDARD_WELD_DATA : WORD ;
    RBT17_STANDARD_WELD_DATA : WORD ;
    RBT18_STANDARD_WELD_DATA : WORD ;
    RBT19_STANDARD_WELD_DATA : WORD ;
    RBT20_STANDARD_WELD_DATA : WORD ;
    RBT21_STANDARD_WELD_DATA : WORD ;
    RBT22_STANDARD_WELD_DATA : WORD ;
    RBT23_STANDARD_WELD_DAT : WORD ;
    RBT24_STANDARD_WELD_DAT : WORD ;
    CHK_WORD : WORD ;
    TEST_TEMP : ARRAY  [1 .. 40 ] OF BYTE ;
   END_STRUCT ;
   S707_BT_CODE_2103 : STRUCT
    STATION_MAIN : WORD ;
    DISTINCTION_LH_RH : WORD ;
    STAION_NUMBER : WORD ;
    BODY_TYPE_1ST : WORD ;
    BODY_TYPE_OPTION : WORD ;
    RBT1_STANDARD_WELD_DATA : WORD ;
    RBT2_STANDARD_WELD_DATA : WORD ;
    RBT3_STANDARD_WELD_DATA : WORD ;
    RBT4_STANDARD_WELD_DATA : WORD ;
    RBT5_STANDARD_WELD_DATA : WORD ;
    RBT6_STANDARD_WELD_DATA : WORD ;
    RBT7_STANDARD_WELD_DATA : WORD ;
    RBT8_STANDARD_WELD_DATA : WORD ;
    RBT9_STANDARD_WELD_DATA : WORD ;
    RBT10_STANDARD_WELD_DATA : WORD ;
    RBT11_STANDARD_WELD_DATA : WORD ;
    RBT12_STANDARD_WELD_DATA : WORD ;
    RBT13_STANDARD_WELD_DATA : WORD ;
    RBT14_STANDARD_WELD_DATA : WORD ;
    RBT15_STANDARD_WELD_DATA : WORD ;
    RBT16_STANDARD_WELD_DATA : WORD ;
    RBT17_STANDARD_WELD_DATA : WORD ;
    RBT18_STANDARD_WELD_DATA : WORD ;
    RBT19_STANDARD_WELD_DATA : WORD ;
    RBT20_STANDARD_WELD_DATA : WORD ;
    RBT21_STANDARD_WELD_DATA : WORD ;
    RBT22_STANDARD_WELD_DATA : WORD ;
    RBT23_STANDARD_WELD_DAT : WORD ;
    RBT24_STANDARD_WELD_DAT : WORD ;
    CHK_WORD : WORD ;
    TEST_TEMP : ARRAY  [1 .. 40 ] OF BYTE ;
   END_STRUCT ;
   S707_BT_CODE_2104 : STRUCT
    STATION_MAIN : WORD ;
    DISTINCTION_LH_RH : WORD ;
    STAION_NUMBER : WORD ;
    BODY_TYPE_1ST : WORD ;
    BODY_TYPE_OPTION : WORD ;
    RBT1_STANDARD_WELD_DATA : WORD ;
    RBT2_STANDARD_WELD_DATA : WORD ;
    RBT3_STANDARD_WELD_DATA : WORD ;
    RBT4_STANDARD_WELD_DATA : WORD ;
    RBT5_STANDARD_WELD_DATA : WORD ;
    RBT6_STANDARD_WELD_DATA : WORD ;
    RBT7_STANDARD_WELD_DATA : WORD ;
    RBT8_STANDARD_WELD_DATA : WORD ;
    RBT9_STANDARD_WELD_DATA : WORD ;
    RBT10_STANDARD_WELD_DATA : WORD ;
    RBT11_STANDARD_WELD_DATA : WORD ;
    RBT12_STANDARD_WELD_DATA : WORD ;
    RBT13_STANDARD_WELD_DATA : WORD ;
    RBT14_STANDARD_WELD_DATA : WORD ;
    RBT15_STANDARD_WELD_DATA : WORD ;
    RBT16_STANDARD_WELD_DATA : WORD ;
    RBT17_STANDARD_WELD_DATA : WORD ;
    RBT18_STANDARD_WELD_DATA : WORD ;
    RBT19_STANDARD_WELD_DATA : WORD ;
    RBT20_STANDARD_WELD_DATA : WORD ;
    RBT21_STANDARD_WELD_DATA : WORD ;
    RBT22_STANDARD_WELD_DATA : WORD ;
    RBT23_STANDARD_WELD_DAT : WORD ;
    RBT24_STANDARD_WELD_DAT : WORD ;
    CHK_WORD : WORD ;
    TEST_TEMP : ARRAY  [1 .. 40 ] OF BYTE ;
   END_STRUCT ;
   S707_BT_CODE_2105 : STRUCT
    STATION_MAIN : WORD ;
    DISTINCTION_LH_RH : WORD ;
    STAION_NUMBER : WORD ;
    BODY_TYPE_1ST : WORD ;
    BODY_TYPE_OPTION : WORD ;
    RBT1_STANDARD_WELD_DATA : WORD ;
    RBT2_STANDARD_WELD_DATA : WORD ;
    RBT3_STANDARD_WELD_DATA : WORD ;
    RBT4_STANDARD_WELD_DATA : WORD ;
    RBT5_STANDARD_WELD_DATA : WORD ;
    RBT6_STANDARD_WELD_DATA : WORD ;
    RBT7_STANDARD_WELD_DATA : WORD ;
    RBT8_STANDARD_WELD_DATA : WORD ;
    RBT9_STANDARD_WELD_DATA : WORD ;
    RBT10_STANDARD_WELD_DATA : WORD ;
    RBT11_STANDARD_WELD_DATA : WORD ;
    RBT12_STANDARD_WELD_DATA : WORD ;
    RBT13_STANDARD_WELD_DATA : WORD ;
    RBT14_STANDARD_WELD_DATA : WORD ;
    RBT15_STANDARD_WELD_DATA : WORD ;
    RBT16_STANDARD_WELD_DATA : WORD ;
    RBT17_STANDARD_WELD_DATA : WORD ;
    RBT18_STANDARD_WELD_DATA : WORD ;
    RBT19_STANDARD_WELD_DATA : WORD ;
    RBT20_STANDARD_WELD_DATA : WORD ;
    RBT21_STANDARD_WELD_DATA : WORD ;
    RBT22_STANDARD_WELD_DATA : WORD ;
    RBT23_STANDARD_WELD_DAT : WORD ;
    RBT24_STANDARD_WELD_DAT : WORD ;
    CHK_WORD : WORD ;
    TEST_TEMP : ARRAY  [1 .. 40 ] OF BYTE ;
   END_STRUCT ;
   S707_BT_CODE_2106 : STRUCT
    STATION_MAIN : WORD ;
    DISTINCTION_LH_RH : WORD ;
    STAION_NUMBER : WORD ;
    BODY_TYPE_1ST : WORD ;
    BODY_TYPE_OPTION : WORD ;
    RBT1_STANDARD_WELD_DATA : WORD ;
    RBT2_STANDARD_WELD_DATA : WORD ;
    RBT3_STANDARD_WELD_DATA : WORD ;
    RBT4_STANDARD_WELD_DATA : WORD ;
    RBT5_STANDARD_WELD_DATA : WORD ;
    RBT6_STANDARD_WELD_DATA : WORD ;
    RBT7_STANDARD_WELD_DATA : WORD ;
    RBT8_STANDARD_WELD_DATA : WORD ;
    RBT9_STANDARD_WELD_DATA : WORD ;
    RBT10_STANDARD_WELD_DATA : WORD ;
    RBT11_STANDARD_WELD_DATA : WORD ;
    RBT12_STANDARD_WELD_DATA : WORD ;
    RBT13_STANDARD_WELD_DATA : WORD ;
    RBT14_STANDARD_WELD_DATA : WORD ;
    RBT15_STANDARD_WELD_DATA : WORD ;
    RBT16_STANDARD_WELD_DATA : WORD ;
    RBT17_STANDARD_WELD_DATA : WORD ;
    RBT18_STANDARD_WELD_DATA : WORD ;
    RBT19_STANDARD_WELD_DATA : WORD ;
    RBT20_STANDARD_WELD_DATA : WORD ;
    RBT21_STANDARD_WELD_DATA : WORD ;
    RBT22_STANDARD_WELD_DATA : WORD ;
    RBT23_STANDARD_WELD_DAT : WORD ;
    RBT24_STANDARD_WELD_DAT : WORD ;
    CHK_WORD : WORD ;
    TEST_TEMP : ARRAY  [1 .. 40 ] OF BYTE ;
   END_STRUCT ;
   S707_BT_CODE_2107 : STRUCT
    STATION_MAIN : WORD ;
    DISTINCTION_LH_RH : WORD ;
    STAION_NUMBER : WORD ;
    BODY_TYPE_1ST : WORD ;
    BODY_TYPE_OPTION : WORD ;
    RBT1_STANDARD_WELD_DATA : WORD ;
    RBT2_STANDARD_WELD_DATA : WORD ;
    RBT3_STANDARD_WELD_DATA : WORD ;
    RBT4_STANDARD_WELD_DATA : WORD ;
    RBT5_STANDARD_WELD_DATA : WORD ;
    RBT6_STANDARD_WELD_DATA : WORD ;
    RBT7_STANDARD_WELD_DATA : WORD ;
    RBT8_STANDARD_WELD_DATA : WORD ;
    RBT9_STANDARD_WELD_DATA : WORD ;
    RBT10_STANDARD_WELD_DATA : WORD ;
    RBT11_STANDARD_WELD_DATA : WORD ;
    RBT12_STANDARD_WELD_DATA : WORD ;
    RBT13_STANDARD_WELD_DATA : WORD ;
    RBT14_STANDARD_WELD_DATA : WORD ;
    RBT15_STANDARD_WELD_DATA : WORD ;
    RBT16_STANDARD_WELD_DATA : WORD ;
    RBT17_STANDARD_WELD_DATA : WORD ;
    RBT18_STANDARD_WELD_DATA : WORD ;
    RBT19_STANDARD_WELD_DATA : WORD ;
    RBT20_STANDARD_WELD_DATA : WORD ;
    RBT21_STANDARD_WELD_DATA : WORD ;
    RBT22_STANDARD_WELD_DATA : WORD ;
    RBT23_STANDARD_WELD_DAT : WORD ;
    RBT24_STANDARD_WELD_DAT : WORD ;
    CHK_WORD : WORD ;
    TEST_TEMP : ARRAY  [1 .. 40 ] OF BYTE ;
   END_STRUCT ;
   S707_BT_CODE_2108 : STRUCT
    STATION_MAIN : WORD ;
    DISTINCTION_LH_RH : WORD ;
    STAION_NUMBER : WORD ;
    BODY_TYPE_1ST : WORD ;
    BODY_TYPE_OPTION : WORD ;
    RBT1_STANDARD_WELD_DATA : WORD ;
    RBT2_STANDARD_WELD_DATA : WORD ;
    RBT3_STANDARD_WELD_DATA : WORD ;
    RBT4_STANDARD_WELD_DATA : WORD ;
    RBT5_STANDARD_WELD_DATA : WORD ;
    RBT6_STANDARD_WELD_DATA : WORD ;
    RBT7_STANDARD_WELD_DATA : WORD ;
    RBT8_STANDARD_WELD_DATA : WORD ;
    RBT9_STANDARD_WELD_DATA : WORD ;
    RBT10_STANDARD_WELD_DATA : WORD ;
    RBT11_STANDARD_WELD_DATA : WORD ;
    RBT12_STANDARD_WELD_DATA : WORD ;
    RBT13_STANDARD_WELD_DATA : WORD ;
    RBT14_STANDARD_WELD_DATA : WORD ;
    RBT15_STANDARD_WELD_DATA : WORD ;
    RBT16_STANDARD_WELD_DATA : WORD ;
    RBT17_STANDARD_WELD_DATA : WORD ;
    RBT18_STANDARD_WELD_DATA : WORD ;
    RBT19_STANDARD_WELD_DATA : WORD ;
    RBT20_STANDARD_WELD_DATA : WORD ;
    RBT21_STANDARD_WELD_DATA : WORD ;
    RBT22_STANDARD_WELD_DATA : WORD ;
    RBT23_STANDARD_WELD_DAT : WORD ;
    RBT24_STANDARD_WELD_DAT : WORD ;
    CHK_WORD : WORD ;
    TEST_TEMP : ARRAY  [1 .. 40 ] OF BYTE ;
   END_STRUCT ;
   S707_BT_CODE_2109 : STRUCT
    STATION_MAIN : WORD ;
    DISTINCTION_LH_RH : WORD ;
    STAION_NUMBER : WORD ;
    BODY_TYPE_1ST : WORD ;
    BODY_TYPE_OPTION : WORD ;
    RBT1_STANDARD_WELD_DATA : WORD ;
    RBT2_STANDARD_WELD_DATA : WORD ;
    RBT3_STANDARD_WELD_DATA : WORD ;
    RBT4_STANDARD_WELD_DATA : WORD ;
    RBT5_STANDARD_WELD_DATA : WORD ;
    RBT6_STANDARD_WELD_DATA : WORD ;
    RBT7_STANDARD_WELD_DATA : WORD ;
    RBT8_STANDARD_WELD_DATA : WORD ;
    RBT9_STANDARD_WELD_DATA : WORD ;
    RBT10_STANDARD_WELD_DATA : WORD ;
    RBT11_STANDARD_WELD_DATA : WORD ;
    RBT12_STANDARD_WELD_DATA : WORD ;
    RBT13_STANDARD_WELD_DATA : WORD ;
    RBT14_STANDARD_WELD_DATA : WORD ;
    RBT15_STANDARD_WELD_DATA : WORD ;
    RBT16_STANDARD_WELD_DATA : WORD ;
    RBT17_STANDARD_WELD_DATA : WORD ;
    RBT18_STANDARD_WELD_DATA : WORD ;
    RBT19_STANDARD_WELD_DATA : WORD ;
    RBT20_STANDARD_WELD_DATA : WORD ;
    RBT21_STANDARD_WELD_DATA : WORD ;
    RBT22_STANDARD_WELD_DATA : WORD ;
    RBT23_STANDARD_WELD_DAT : WORD ;
    RBT24_STANDARD_WELD_DAT : WORD ;
    CHK_WORD : WORD ;
    TEST_TEMP : ARRAY  [1 .. 40 ] OF BYTE ;
   END_STRUCT ;
   S707_BT_CODE_2110 : STRUCT
    STATION_MAIN : WORD ;
    DISTINCTION_LH_RH : WORD ;
    STAION_NUMBER : WORD ;
    BODY_TYPE_1ST : WORD ;
    BODY_TYPE_OPTION : WORD ;
    RBT1_STANDARD_WELD_DATA : WORD ;
    RBT2_STANDARD_WELD_DATA : WORD ;
    RBT3_STANDARD_WELD_DATA : WORD ;
    RBT4_STANDARD_WELD_DATA : WORD ;
    RBT5_STANDARD_WELD_DATA : WORD ;
    RBT6_STANDARD_WELD_DATA : WORD ;
    RBT7_STANDARD_WELD_DATA : WORD ;
    RBT8_STANDARD_WELD_DATA : WORD ;
    RBT9_STANDARD_WELD_DATA : WORD ;
    RBT10_STANDARD_WELD_DATA : WORD ;
    RBT11_STANDARD_WELD_DATA : WORD ;
    RBT12_STANDARD_WELD_DATA : WORD ;
    RBT13_STANDARD_WELD_DATA : WORD ;
    RBT14_STANDARD_WELD_DATA : WORD ;
    RBT15_STANDARD_WELD_DATA : WORD ;
    RBT16_STANDARD_WELD_DATA : WORD ;
    RBT17_STANDARD_WELD_DATA : WORD ;
    RBT18_STANDARD_WELD_DATA : WORD ;
    RBT19_STANDARD_WELD_DATA : WORD ;
    RBT20_STANDARD_WELD_DATA : WORD ;
    RBT21_STANDARD_WELD_DATA : WORD ;
    RBT22_STANDARD_WELD_DATA : WORD ;
    RBT23_STANDARD_WELD_DAT : WORD ;
    RBT24_STANDARD_WELD_DAT : WORD ;
    CHK_WORD : WORD ;
    TEST_TEMP : ARRAY  [1 .. 40 ] OF BYTE ;
   END_STRUCT ;
   S707_BT_CODE_2111 : STRUCT
    STATION_MAIN : WORD ;
    DISTINCTION_LH_RH : WORD ;
    STAION_NUMBER : WORD ;
    BODY_TYPE_1ST : WORD ;
    BODY_TYPE_OPTION : WORD ;
    RBT1_STANDARD_WELD_DATA : WORD ;
    RBT2_STANDARD_WELD_DATA : WORD ;
    RBT3_STANDARD_WELD_DATA : WORD ;
    RBT4_STANDARD_WELD_DATA : WORD ;
    RBT5_STANDARD_WELD_DATA : WORD ;
    RBT6_STANDARD_WELD_DATA : WORD ;
    RBT7_STANDARD_WELD_DATA : WORD ;
    RBT8_STANDARD_WELD_DATA : WORD ;
    RBT9_STANDARD_WELD_DATA : WORD ;
    RBT10_STANDARD_WELD_DATA : WORD ;
    RBT11_STANDARD_WELD_DATA : WORD ;
    RBT12_STANDARD_WELD_DATA : WORD ;
    RBT13_STANDARD_WELD_DATA : WORD ;
    RBT14_STANDARD_WELD_DATA : WORD ;
    RBT15_STANDARD_WELD_DATA : WORD ;
    RBT16_STANDARD_WELD_DATA : WORD ;
    RBT17_STANDARD_WELD_DATA : WORD ;
    RBT18_STANDARD_WELD_DATA : WORD ;
    RBT19_STANDARD_WELD_DATA : WORD ;
    RBT20_STANDARD_WELD_DATA : WORD ;
    RBT21_STANDARD_WELD_DATA : WORD ;
    RBT22_STANDARD_WELD_DATA : WORD ;
    RBT23_STANDARD_WELD_DAT : WORD ;
    RBT24_STANDARD_WELD_DAT : WORD ;
    CHK_WORD : WORD ;
    TEST_TEMP : ARRAY  [1 .. 40 ] OF BYTE ;
   END_STRUCT ;
   S707_BT_CODE_2112 : STRUCT
    STATION_MAIN : WORD ;
    DISTINCTION_LH_RH : WORD ;
    STAION_NUMBER : WORD ;
    BODY_TYPE_1ST : WORD ;
    BODY_TYPE_OPTION : WORD ;
    RBT1_STANDARD_WELD_DATA : WORD ;
    RBT2_STANDARD_WELD_DATA : WORD ;
    RBT3_STANDARD_WELD_DATA : WORD ;
    RBT4_STANDARD_WELD_DATA : WORD ;
    RBT5_STANDARD_WELD_DATA : WORD ;
    RBT6_STANDARD_WELD_DATA : WORD ;
    RBT7_STANDARD_WELD_DATA : WORD ;
    RBT8_STANDARD_WELD_DATA : WORD ;
    RBT9_STANDARD_WELD_DATA : WORD ;
    RBT10_STANDARD_WELD_DATA : WORD ;
    RBT11_STANDARD_WELD_DATA : WORD ;
    RBT12_STANDARD_WELD_DATA : WORD ;
    RBT13_STANDARD_WELD_DATA : WORD ;
    RBT14_STANDARD_WELD_DATA : WORD ;
    RBT15_STANDARD_WELD_DATA : WORD ;
    RBT16_STANDARD_WELD_DATA : WORD ;
    RBT17_STANDARD_WELD_DATA : WORD ;
    RBT18_STANDARD_WELD_DATA : WORD ;
    RBT19_STANDARD_WELD_DATA : WORD ;
    RBT20_STANDARD_WELD_DATA : WORD ;
    RBT21_STANDARD_WELD_DATA : WORD ;
    RBT22_STANDARD_WELD_DATA : WORD ;
    RBT23_STANDARD_WELD_DAT : WORD ;
    RBT24_STANDARD_WELD_DAT : WORD ;
    CHK_WORD : WORD ;
    TEST_TEMP : ARRAY  [1 .. 40 ] OF BYTE ;
   END_STRUCT ;
   S707_BT_CODE_2113 : STRUCT
    STATION_MAIN : WORD ;
    DISTINCTION_LH_RH : WORD ;
    STAION_NUMBER : WORD ;
    BODY_TYPE_1ST : WORD ;
    BODY_TYPE_OPTION : WORD ;
    RBT1_STANDARD_WELD_DATA : WORD ;
    RBT2_STANDARD_WELD_DATA : WORD ;
    RBT3_STANDARD_WELD_DATA : WORD ;
    RBT4_STANDARD_WELD_DATA : WORD ;
    RBT5_STANDARD_WELD_DATA : WORD ;
    RBT6_STANDARD_WELD_DATA : WORD ;
    RBT7_STANDARD_WELD_DATA : WORD ;
    RBT8_STANDARD_WELD_DATA : WORD ;
    RBT9_STANDARD_WELD_DATA : WORD ;
    RBT10_STANDARD_WELD_DATA : WORD ;
    RBT11_STANDARD_WELD_DATA : WORD ;
    RBT12_STANDARD_WELD_DATA : WORD ;
    RBT13_STANDARD_WELD_DATA : WORD ;
    RBT14_STANDARD_WELD_DATA : WORD ;
    RBT15_STANDARD_WELD_DATA : WORD ;
    RBT16_STANDARD_WELD_DATA : WORD ;
    RBT17_STANDARD_WELD_DATA : WORD ;
    RBT18_STANDARD_WELD_DATA : WORD ;
    RBT19_STANDARD_WELD_DATA : WORD ;
    RBT20_STANDARD_WELD_DATA : WORD ;
    RBT21_STANDARD_WELD_DATA : WORD ;
    RBT22_STANDARD_WELD_DATA : WORD ;
    RBT23_STANDARD_WELD_DAT : WORD ;
    RBT24_STANDARD_WELD_DAT : WORD ;
    CHK_WORD : WORD ;
    TEST_TEMP : ARRAY  [1 .. 40 ] OF BYTE ;
   END_STRUCT ;
   S707_BT_CODE_2114 : STRUCT
    STATION_MAIN : WORD ;
    DISTINCTION_LH_RH : WORD ;
    STAION_NUMBER : WORD ;
    BODY_TYPE_1ST : WORD ;
    BODY_TYPE_OPTION : WORD ;
    RBT1_STANDARD_WELD_DATA : WORD ;
    RBT2_STANDARD_WELD_DATA : WORD ;
    RBT3_STANDARD_WELD_DATA : WORD ;
    RBT4_STANDARD_WELD_DATA : WORD ;
    RBT5_STANDARD_WELD_DATA : WORD ;
    RBT6_STANDARD_WELD_DATA : WORD ;
    RBT7_STANDARD_WELD_DATA : WORD ;
    RBT8_STANDARD_WELD_DATA : WORD ;
    RBT9_STANDARD_WELD_DATA : WORD ;
    RBT10_STANDARD_WELD_DATA : WORD ;
    RBT11_STANDARD_WELD_DATA : WORD ;
    RBT12_STANDARD_WELD_DATA : WORD ;
    RBT13_STANDARD_WELD_DATA : WORD ;
    RBT14_STANDARD_WELD_DATA : WORD ;
    RBT15_STANDARD_WELD_DATA : WORD ;
    RBT16_STANDARD_WELD_DATA : WORD ;
    RBT17_STANDARD_WELD_DATA : WORD ;
    RBT18_STANDARD_WELD_DATA : WORD ;
    RBT19_STANDARD_WELD_DATA : WORD ;
    RBT20_STANDARD_WELD_DATA : WORD ;
    RBT21_STANDARD_WELD_DATA : WORD ;
    RBT22_STANDARD_WELD_DATA : WORD ;
    RBT23_STANDARD_WELD_DAT : WORD ;
    RBT24_STANDARD_WELD_DAT : WORD ;
    CHK_WORD : WORD ;
    TEST_TEMP : ARRAY  [1 .. 40 ] OF BYTE ;
   END_STRUCT ;
   S707_BT_CODE_2115 : STRUCT
    STATION_MAIN : WORD ;
    DISTINCTION_LH_RH : WORD ;
    STAION_NUMBER : WORD ;
    BODY_TYPE_1ST : WORD ;
    BODY_TYPE_OPTION : WORD ;
    RBT1_STANDARD_WELD_DATA : WORD ;
    RBT2_STANDARD_WELD_DATA : WORD ;
    RBT3_STANDARD_WELD_DATA : WORD ;
    RBT4_STANDARD_WELD_DATA : WORD ;
    RBT5_STANDARD_WELD_DATA : WORD ;
    RBT6_STANDARD_WELD_DATA : WORD ;
    RBT7_STANDARD_WELD_DATA : WORD ;
    RBT8_STANDARD_WELD_DATA : WORD ;
    RBT9_STANDARD_WELD_DATA : WORD ;
    RBT10_STANDARD_WELD_DATA : WORD ;
    RBT11_STANDARD_WELD_DATA : WORD ;
    RBT12_STANDARD_WELD_DATA : WORD ;
    RBT13_STANDARD_WELD_DATA : WORD ;
    RBT14_STANDARD_WELD_DATA : WORD ;
    RBT15_STANDARD_WELD_DATA : WORD ;
    RBT16_STANDARD_WELD_DATA : WORD ;
    RBT17_STANDARD_WELD_DATA : WORD ;
    RBT18_STANDARD_WELD_DATA : WORD ;
    RBT19_STANDARD_WELD_DATA : WORD ;
    RBT20_STANDARD_WELD_DATA : WORD ;
    RBT21_STANDARD_WELD_DATA : WORD ;
    RBT22_STANDARD_WELD_DATA : WORD ;
    RBT23_STANDARD_WELD_DAT : WORD ;
    RBT24_STANDARD_WELD_DAT : WORD ;
    CHK_WORD : WORD ;
    TEST_TEMP : ARRAY  [1 .. 40 ] OF BYTE ;
   END_STRUCT ;
   S707_BT_CODE_2116 : STRUCT
    STATION_MAIN : WORD ;
    DISTINCTION_LH_RH : WORD ;
    STAION_NUMBER : WORD ;
    BODY_TYPE_1ST : WORD ;
    BODY_TYPE_OPTION : WORD ;
    RBT1_STANDARD_WELD_DATA : WORD ;
    RBT2_STANDARD_WELD_DATA : WORD ;
    RBT3_STANDARD_WELD_DATA : WORD ;
    RBT4_STANDARD_WELD_DATA : WORD ;
    RBT5_STANDARD_WELD_DATA : WORD ;
    RBT6_STANDARD_WELD_DATA : WORD ;
    RBT7_STANDARD_WELD_DATA : WORD ;
    RBT8_STANDARD_WELD_DATA : WORD ;
    RBT9_STANDARD_WELD_DATA : WORD ;
    RBT10_STANDARD_WELD_DATA : WORD ;
    RBT11_STANDARD_WELD_DATA : WORD ;
    RBT12_STANDARD_WELD_DATA : WORD ;
    RBT13_STANDARD_WELD_DATA : WORD ;
    RBT14_STANDARD_WELD_DATA : WORD ;
    RBT15_STANDARD_WELD_DATA : WORD ;
    RBT16_STANDARD_WELD_DATA : WORD ;
    RBT17_STANDARD_WELD_DATA : WORD ;
    RBT18_STANDARD_WELD_DATA : WORD ;
    RBT19_STANDARD_WELD_DATA : WORD ;
    RBT20_STANDARD_WELD_DATA : WORD ;
    RBT21_STANDARD_WELD_DATA : WORD ;
    RBT22_STANDARD_WELD_DATA : WORD ;
    RBT23_STANDARD_WELD_DAT : WORD ;
    RBT24_STANDARD_WELD_DAT : WORD ;
    CHK_WORD : WORD ;
    TEST_TEMP : ARRAY  [1 .. 40 ] OF BYTE ;
   END_STRUCT ;
   S707_BT_CODE_2117 : STRUCT
    STATION_MAIN : WORD ;
    DISTINCTION_LH_RH : WORD ;
    STAION_NUMBER : WORD ;
    BODY_TYPE_1ST : WORD ;
    BODY_TYPE_OPTION : WORD ;
    RBT1_STANDARD_WELD_DATA : WORD ;
    RBT2_STANDARD_WELD_DATA : WORD ;
    RBT3_STANDARD_WELD_DATA : WORD ;
    RBT4_STANDARD_WELD_DATA : WORD ;
    RBT5_STANDARD_WELD_DATA : WORD ;
    RBT6_STANDARD_WELD_DATA : WORD ;
    RBT7_STANDARD_WELD_DATA : WORD ;
    RBT8_STANDARD_WELD_DATA : WORD ;
    RBT9_STANDARD_WELD_DATA : WORD ;
    RBT10_STANDARD_WELD_DATA : WORD ;
    RBT11_STANDARD_WELD_DATA : WORD ;
    RBT12_STANDARD_WELD_DATA : WORD ;
    RBT13_STANDARD_WELD_DATA : WORD ;
    RBT14_STANDARD_WELD_DATA : WORD ;
    RBT15_STANDARD_WELD_DATA : WORD ;
    RBT16_STANDARD_WELD_DATA : WORD ;
    RBT17_STANDARD_WELD_DATA : WORD ;
    RBT18_STANDARD_WELD_DATA : WORD ;
    RBT19_STANDARD_WELD_DATA : WORD ;
    RBT20_STANDARD_WELD_DATA : WORD ;
    RBT21_STANDARD_WELD_DATA : WORD ;
    RBT22_STANDARD_WELD_DATA : WORD ;
    RBT23_STANDARD_WELD_DAT : WORD ;
    RBT24_STANDARD_WELD_DAT : WORD ;
    CHK_WORD : WORD ;
    TEST_TEMP : ARRAY  [1 .. 40 ] OF BYTE ;
   END_STRUCT ;
   S707_BT_CODE_2118 : STRUCT
    STATION_MAIN : WORD ;
    DISTINCTION_LH_RH : WORD ;
    STAION_NUMBER : WORD ;
    BODY_TYPE_1ST : WORD ;
    BODY_TYPE_OPTION : WORD ;
    RBT1_STANDARD_WELD_DATA : WORD ;
    RBT2_STANDARD_WELD_DATA : WORD ;
    RBT3_STANDARD_WELD_DATA : WORD ;
    RBT4_STANDARD_WELD_DATA : WORD ;
    RBT5_STANDARD_WELD_DATA : WORD ;
    RBT6_STANDARD_WELD_DATA : WORD ;
    RBT7_STANDARD_WELD_DATA : WORD ;
    RBT8_STANDARD_WELD_DATA : WORD ;
    RBT9_STANDARD_WELD_DATA : WORD ;
    RBT10_STANDARD_WELD_DATA : WORD ;
    RBT11_STANDARD_WELD_DATA : WORD ;
    RBT12_STANDARD_WELD_DATA : WORD ;
    RBT13_STANDARD_WELD_DATA : WORD ;
    RBT14_STANDARD_WELD_DATA : WORD ;
    RBT15_STANDARD_WELD_DATA : WORD ;
    RBT16_STANDARD_WELD_DATA : WORD ;
    RBT17_STANDARD_WELD_DATA : WORD ;
    RBT18_STANDARD_WELD_DATA : WORD ;
    RBT19_STANDARD_WELD_DATA : WORD ;
    RBT20_STANDARD_WELD_DATA : WORD ;
    RBT21_STANDARD_WELD_DATA : WORD ;
    RBT22_STANDARD_WELD_DATA : WORD ;
    RBT23_STANDARD_WELD_DAT : WORD ;
    RBT24_STANDARD_WELD_DAT : WORD ;
    CHK_WORD : WORD ;
    TEST_TEMP : ARRAY  [1 .. 40 ] OF BYTE ;
   END_STRUCT ;
   S707_BT_CODE_2119 : STRUCT
    STATION_MAIN : WORD ;
    DISTINCTION_LH_RH : WORD ;
    STAION_NUMBER : WORD ;
    BODY_TYPE_1ST : WORD ;
    BODY_TYPE_OPTION : WORD ;
    RBT1_STANDARD_WELD_DATA : WORD ;
    RBT2_STANDARD_WELD_DATA : WORD ;
    RBT3_STANDARD_WELD_DATA : WORD ;
    RBT4_STANDARD_WELD_DATA : WORD ;
    RBT5_STANDARD_WELD_DATA : WORD ;
    RBT6_STANDARD_WELD_DATA : WORD ;
    RBT7_STANDARD_WELD_DATA : WORD ;
    RBT8_STANDARD_WELD_DATA : WORD ;
    RBT9_STANDARD_WELD_DATA : WORD ;
    RBT10_STANDARD_WELD_DATA : WORD ;
    RBT11_STANDARD_WELD_DATA : WORD ;
    RBT12_STANDARD_WELD_DATA : WORD ;
    RBT13_STANDARD_WELD_DATA : WORD ;
    RBT14_STANDARD_WELD_DATA : WORD ;
    RBT15_STANDARD_WELD_DATA : WORD ;
    RBT16_STANDARD_WELD_DATA : WORD ;
    RBT17_STANDARD_WELD_DATA : WORD ;
    RBT18_STANDARD_WELD_DATA : WORD ;
    RBT19_STANDARD_WELD_DATA : WORD ;
    RBT20_STANDARD_WELD_DATA : WORD ;
    RBT21_STANDARD_WELD_DATA : WORD ;
    RBT22_STANDARD_WELD_DATA : WORD ;
    RBT23_STANDARD_WELD_DAT : WORD ;
    RBT24_STANDARD_WELD_DAT : WORD ;
    CHK_WORD : WORD ;
    TEST_TEMP : ARRAY  [1 .. 40 ] OF BYTE ;
   END_STRUCT ;
   S707_BT_CODE_2120 : STRUCT
    STATION_MAIN : WORD ;
    DISTINCTION_LH_RH : WORD ;
    STAION_NUMBER : WORD ;
    BODY_TYPE_1ST : WORD ;
    BODY_TYPE_OPTION : WORD ;
    RBT1_STANDARD_WELD_DATA : WORD ;
    RBT2_STANDARD_WELD_DATA : WORD ;
    RBT3_STANDARD_WELD_DATA : WORD ;
    RBT4_STANDARD_WELD_DATA : WORD ;
    RBT5_STANDARD_WELD_DATA : WORD ;
    RBT6_STANDARD_WELD_DATA : WORD ;
    RBT7_STANDARD_WELD_DATA : WORD ;
    RBT8_STANDARD_WELD_DATA : WORD ;
    RBT9_STANDARD_WELD_DATA : WORD ;
    RBT10_STANDARD_WELD_DATA : WORD ;
    RBT11_STANDARD_WELD_DATA : WORD ;
    RBT12_STANDARD_WELD_DATA : WORD ;
    RBT13_STANDARD_WELD_DATA : WORD ;
    RBT14_STANDARD_WELD_DATA : WORD ;
    RBT15_STANDARD_WELD_DATA : WORD ;
    RBT16_STANDARD_WELD_DATA : WORD ;
    RBT17_STANDARD_WELD_DATA : WORD ;
    RBT18_STANDARD_WELD_DATA : WORD ;
    RBT19_STANDARD_WELD_DATA : WORD ;
    RBT20_STANDARD_WELD_DATA : WORD ;
    RBT21_STANDARD_WELD_DATA : WORD ;
    RBT22_STANDARD_WELD_DATA : WORD ;
    RBT23_STANDARD_WELD_DAT : WORD ;
    RBT24_STANDARD_WELD_DAT : WORD ;
    CHK_WORD : WORD ;
    TEST_TEMP : ARRAY  [1 .. 40 ] OF BYTE ;
   END_STRUCT ;
  END_STRUCT ;
BEGIN
   S705_BT_CODE_2011.STATION_MAIN := W#16#2C1;
   S705_BT_CODE_2011.DISTINCTION_LH_RH := W#16#1;
   S705_BT_CODE_2011.STAION_NUMBER := W#16#0;
   S705_BT_CODE_2011.BODY_TYPE_1ST := W#16#1;
   S705_BT_CODE_2011.BODY_TYPE_OPTION := W#16#7DB;
   S705_BT_CODE_2011.RBT1_STANDARD_WELD_DATA := W#16#3;
   S705_BT_CODE_2011.RBT2_STANDARD_WELD_DATA := W#16#0;
   S705_BT_CODE_2011.RBT3_STANDARD_WELD_DATA := W#16#0;
   S705_BT_CODE_2011.RBT4_STANDARD_WELD_DATA := W#16#0;
   S705_BT_CODE_2011.RBT5_STANDARD_WELD_DATA := W#16#0;
   S705_BT_CODE_2011.RBT6_STANDARD_WELD_DATA := W#16#0;
   S705_BT_CODE_2011.RBT7_STANDARD_WELD_DATA := W#16#0;
   S705_BT_CODE_2011.RBT8_STANDARD_WELD_DATA := W#16#0;
   S705_BT_CODE_2011.RBT9_STANDARD_WELD_DATA := W#16#0;
   S705_BT_CODE_2011.RBT10_STANDARD_WELD_DATA := W#16#0;
   S705_BT_CODE_2011.RBT11_STANDARD_WELD_DATA := W#16#0;
   S705_BT_CODE_2011.RBT12_STANDARD_WELD_DATA := W#16#0;
   S705_BT_CODE_2011.RBT13_STANDARD_WELD_DATA := W#16#0;
   S705_BT_CODE_2011.RBT14_STANDARD_WELD_DATA := W#16#0;
   S705_BT_CODE_2011.RBT15_STANDARD_WELD_DATA := W#16#0;
   S705_BT_CODE_2011.RBT16_STANDARD_WELD_DATA := W#16#0;
   S705_BT_CODE_2011.RBT17_STANDARD_WELD_DATA := W#16#0;
   S705_BT_CODE_2011.RBT18_STANDARD_WELD_DATA := W#16#0;
   S705_BT_CODE_2011.RBT19_STANDARD_WELD_DATA := W#16#0;
   S705_BT_CODE_2011.RBT20_STANDARD_WELD_DATA := W#16#0;
   S705_BT_CODE_2011.RBT21_STANDARD_WELD_DATA := W#16#0;
   S705_BT_CODE_2011.RBT22_STANDARD_WELD_DATA := W#16#0;
   S705_BT_CODE_2011.RBT23_STANDARD_WELD_DAT := W#16#0;
   S705_BT_CODE_2011.RBT24_STANDARD_WELD_DAT := W#16#0;
   S705_BT_CODE_2011.CHK_WORD := W#16#0;
   S705_BT_CODE_2011.TEST_TEMP[1] := B#16#0;
   S705_BT_CODE_2011.TEST_TEMP[2] := B#16#0;
   S705_BT_CODE_2011.TEST_TEMP[3] := B#16#0;
   S705_BT_CODE_2011.TEST_TEMP[4] := B#16#0;
   S705_BT_CODE_2011.TEST_TEMP[5] := B#16#0;
   S705_BT_CODE_2011.TEST_TEMP[6] := B#16#0;
   S705_BT_CODE_2011.TEST_TEMP[7] := B#16#0;
   S705_BT_CODE_2011.TEST_TEMP[8] := B#16#0;
   S705_BT_CODE_2011.TEST_TEMP[9] := B#16#0;
   S705_BT_CODE_2011.TEST_TEMP[10] := B#16#0;
   S705_BT_CODE_2011.TEST_TEMP[11] := B#16#0;
   S705_BT_CODE_2011.TEST_TEMP[12] := B#16#0;
   S705_BT_CODE_2011.TEST_TEMP[13] := B#16#0;
   S705_BT_CODE_2011.TEST_TEMP[14] := B#16#0;
   S705_BT_CODE_2011.TEST_TEMP[15] := B#16#0;
   S705_BT_CODE_2011.TEST_TEMP[16] := B#16#0;
   S705_BT_CODE_2011.TEST_TEMP[17] := B#16#0;
   S705_BT_CODE_2011.TEST_TEMP[18] := B#16#0;
   S705_BT_CODE_2011.TEST_TEMP[19] := B#16#0;
   S705_BT_CODE_2011.TEST_TEMP[20] := B#16#0;
   S705_BT_CODE_2011.TEST_TEMP[21] := B#16#0;
   S705_BT_CODE_2011.TEST_TEMP[22] := B#16#0;
   S705_BT_CODE_2011.TEST_TEMP[23] := B#16#0;
   S705_BT_CODE_2011.TEST_TEMP[24] := B#16#0;
   S705_BT_CODE_2011.TEST_TEMP[25] := B#16#0;
   S705_BT_CODE_2011.TEST_TEMP[26] := B#16#0;
   S705_BT_CODE_2011.TEST_TEMP[27] := B#16#0;
   S705_BT_CODE_2011.TEST_TEMP[28] := B#16#0;
   S705_BT_CODE_2011.TEST_TEMP[29] := B#16#0;
   S705_BT_CODE_2011.TEST_TEMP[30] := B#16#0;
   S705_BT_CODE_2011.TEST_TEMP[31] := B#16#0;
   S705_BT_CODE_2011.TEST_TEMP[32] := B#16#0;
   S705_BT_CODE_2011.TEST_TEMP[33] := B#16#0;
   S705_BT_CODE_2011.TEST_TEMP[34] := B#16#0;
   S705_BT_CODE_2011.TEST_TEMP[35] := B#16#0;
   S705_BT_CODE_2011.TEST_TEMP[36] := B#16#0;
   S705_BT_CODE_2011.TEST_TEMP[37] := B#16#0;
   S705_BT_CODE_2011.TEST_TEMP[38] := B#16#0;
   S705_BT_CODE_2011.TEST_TEMP[39] := B#16#0;
   S705_BT_CODE_2011.TEST_TEMP[40] := B#16#0;
   S705_BT_CODE_2012.STATION_MAIN := W#16#0;
   S705_BT_CODE_2012.DISTINCTION_LH_RH := W#16#0;
   S705_BT_CODE_2012.STAION_NUMBER := W#16#0;
   S705_BT_CODE_2012.BODY_TYPE_1ST := W#16#0;
   S705_BT_CODE_2012.BODY_TYPE_OPTION := W#16#0;
   S705_BT_CODE_2012.RBT1_STANDARD_WELD_DATA := W#16#0;
   S705_BT_CODE_2012.RBT2_STANDARD_WELD_DATA := W#16#0;
   S705_BT_CODE_2012.RBT3_STANDARD_WELD_DATA := W#16#0;
   S705_BT_CODE_2012.RBT4_STANDARD_WELD_DATA := W#16#0;
   S705_BT_CODE_2012.RBT5_STANDARD_WELD_DATA := W#16#0;
   S705_BT_CODE_2012.RBT6_STANDARD_WELD_DATA := W#16#0;
   S705_BT_CODE_2012.RBT7_STANDARD_WELD_DATA := W#16#0;
   S705_BT_CODE_2012.RBT8_STANDARD_WELD_DATA := W#16#0;
   S705_BT_CODE_2012.RBT9_STANDARD_WELD_DATA := W#16#0;
   S705_BT_CODE_2012.RBT10_STANDARD_WELD_DATA := W#16#0;
   S705_BT_CODE_2012.RBT11_STANDARD_WELD_DATA := W#16#0;
   S705_BT_CODE_2012.RBT12_STANDARD_WELD_DATA := W#16#0;
   S705_BT_CODE_2012.RBT13_STANDARD_WELD_DATA := W#16#0;
   S705_BT_CODE_2012.RBT14_STANDARD_WELD_DATA := W#16#0;
   S705_BT_CODE_2012.RBT15_STANDARD_WELD_DATA := W#16#0;
   S705_BT_CODE_2012.RBT16_STANDARD_WELD_DATA := W#16#0;
   S705_BT_CODE_2012.RBT17_STANDARD_WELD_DATA := W#16#0;
   S705_BT_CODE_2012.RBT18_STANDARD_WELD_DATA := W#16#0;
   S705_BT_CODE_2012.RBT19_STANDARD_WELD_DATA := W#16#0;
   S705_BT_CODE_2012.RBT20_STANDARD_WELD_DATA := W#16#0;
   S705_BT_CODE_2012.RBT21_STANDARD_WELD_DATA := W#16#0;
   S705_BT_CODE_2012.RBT22_STANDARD_WELD_DATA := W#16#0;
   S705_BT_CODE_2012.RBT23_STANDARD_WELD_DAT := W#16#0;
   S705_BT_CODE_2012.RBT24_STANDARD_WELD_DAT := W#16#0;
   S705_BT_CODE_2012.CHK_WORD := W#16#0;
   S705_BT_CODE_2012.TEST_TEMP[1] := B#16#0;
   S705_BT_CODE_2012.TEST_TEMP[2] := B#16#0;
   S705_BT_CODE_2012.TEST_TEMP[3] := B#16#0;
   S705_BT_CODE_2012.TEST_TEMP[4] := B#16#0;
   S705_BT_CODE_2012.TEST_TEMP[5] := B#16#0;
   S705_BT_CODE_2012.TEST_TEMP[6] := B#16#0;
   S705_BT_CODE_2012.TEST_TEMP[7] := B#16#0;
   S705_BT_CODE_2012.TEST_TEMP[8] := B#16#0;
   S705_BT_CODE_2012.TEST_TEMP[9] := B#16#0;
   S705_BT_CODE_2012.TEST_TEMP[10] := B#16#0;
   S705_BT_CODE_2012.TEST_TEMP[11] := B#16#0;
   S705_BT_CODE_2012.TEST_TEMP[12] := B#16#0;
   S705_BT_CODE_2012.TEST_TEMP[13] := B#16#0;
   S705_BT_CODE_2012.TEST_TEMP[14] := B#16#0;
   S705_BT_CODE_2012.TEST_TEMP[15] := B#16#0;
   S705_BT_CODE_2012.TEST_TEMP[16] := B#16#0;
   S705_BT_CODE_2012.TEST_TEMP[17] := B#16#0;
   S705_BT_CODE_2012.TEST_TEMP[18] := B#16#0;
   S705_BT_CODE_2012.TEST_TEMP[19] := B#16#0;
   S705_BT_CODE_2012.TEST_TEMP[20] := B#16#0;
   S705_BT_CODE_2012.TEST_TEMP[21] := B#16#0;
   S705_BT_CODE_2012.TEST_TEMP[22] := B#16#0;
   S705_BT_CODE_2012.TEST_TEMP[23] := B#16#0;
   S705_BT_CODE_2012.TEST_TEMP[24] := B#16#0;
   S705_BT_CODE_2012.TEST_TEMP[25] := B#16#0;
   S705_BT_CODE_2012.TEST_TEMP[26] := B#16#0;
   S705_BT_CODE_2012.TEST_TEMP[27] := B#16#0;
   S705_BT_CODE_2012.TEST_TEMP[28] := B#16#0;
   S705_BT_CODE_2012.TEST_TEMP[29] := B#16#0;
   S705_BT_CODE_2012.TEST_TEMP[30] := B#16#0;
   S705_BT_CODE_2012.TEST_TEMP[31] := B#16#0;
   S705_BT_CODE_2012.TEST_TEMP[32] := B#16#0;
   S705_BT_CODE_2012.TEST_TEMP[33] := B#16#0;
   S705_BT_CODE_2012.TEST_TEMP[34] := B#16#0;
   S705_BT_CODE_2012.TEST_TEMP[35] := B#16#0;
   S705_BT_CODE_2012.TEST_TEMP[36] := B#16#0;
   S705_BT_CODE_2012.TEST_TEMP[37] := B#16#0;
   S705_BT_CODE_2012.TEST_TEMP[38] := B#16#0;
   S705_BT_CODE_2012.TEST_TEMP[39] := B#16#0;
   S705_BT_CODE_2012.TEST_TEMP[40] := B#16#0;
   S705_BT_CODE_2013.STATION_MAIN := W#16#0;
   S705_BT_CODE_2013.DISTINCTION_LH_RH := W#16#0;
   S705_BT_CODE_2013.STAION_NUMBER := W#16#0;
   S705_BT_CODE_2013.BODY_TYPE_1ST := W#16#0;
   S705_BT_CODE_2013.BODY_TYPE_OPTION := W#16#0;
   S705_BT_CODE_2013.RBT1_STANDARD_WELD_DATA := W#16#0;
   S705_BT_CODE_2013.RBT2_STANDARD_WELD_DATA := W#16#0;
   S705_BT_CODE_2013.RBT3_STANDARD_WELD_DATA := W#16#0;
   S705_BT_CODE_2013.RBT4_STANDARD_WELD_DATA := W#16#0;
   S705_BT_CODE_2013.RBT5_STANDARD_WELD_DATA := W#16#0;
   S705_BT_CODE_2013.RBT6_STANDARD_WELD_DATA := W#16#0;
   S705_BT_CODE_2013.RBT7_STANDARD_WELD_DATA := W#16#0;
   S705_BT_CODE_2013.RBT8_STANDARD_WELD_DATA := W#16#0;
   S705_BT_CODE_2013.RBT9_STANDARD_WELD_DATA := W#16#0;
   S705_BT_CODE_2013.RBT10_STANDARD_WELD_DATA := W#16#0;
   S705_BT_CODE_2013.RBT11_STANDARD_WELD_DATA := W#16#0;
   S705_BT_CODE_2013.RBT12_STANDARD_WELD_DATA := W#16#0;
   S705_BT_CODE_2013.RBT13_STANDARD_WELD_DATA := W#16#0;
   S705_BT_CODE_2013.RBT14_STANDARD_WELD_DATA := W#16#0;
   S705_BT_CODE_2013.RBT15_STANDARD_WELD_DATA := W#16#0;
   S705_BT_CODE_2013.RBT16_STANDARD_WELD_DATA := W#16#0;
   S705_BT_CODE_2013.RBT17_STANDARD_WELD_DATA := W#16#0;
   S705_BT_CODE_2013.RBT18_STANDARD_WELD_DATA := W#16#0;
   S705_BT_CODE_2013.RBT19_STANDARD_WELD_DATA := W#16#0;
   S705_BT_CODE_2013.RBT20_STANDARD_WELD_DATA := W#16#0;
   S705_BT_CODE_2013.RBT21_STANDARD_WELD_DATA := W#16#0;
   S705_BT_CODE_2013.RBT22_STANDARD_WELD_DATA := W#16#0;
   S705_BT_CODE_2013.RBT23_STANDARD_WELD_DAT := W#16#0;
   S705_BT_CODE_2013.RBT24_STANDARD_WELD_DAT := W#16#0;
   S705_BT_CODE_2013.CHK_WORD := W#16#0;
   S705_BT_CODE_2013.TEST_TEMP[1] := B#16#0;
   S705_BT_CODE_2013.TEST_TEMP[2] := B#16#0;
   S705_BT_CODE_2013.TEST_TEMP[3] := B#16#0;
   S705_BT_CODE_2013.TEST_TEMP[4] := B#16#0;
   S705_BT_CODE_2013.TEST_TEMP[5] := B#16#0;
   S705_BT_CODE_2013.TEST_TEMP[6] := B#16#0;
   S705_BT_CODE_2013.TEST_TEMP[7] := B#16#0;
   S705_BT_CODE_2013.TEST_TEMP[8] := B#16#0;
   S705_BT_CODE_2013.TEST_TEMP[9] := B#16#0;
   S705_BT_CODE_2013.TEST_TEMP[10] := B#16#0;
   S705_BT_CODE_2013.TEST_TEMP[11] := B#16#0;
   S705_BT_CODE_2013.TEST_TEMP[12] := B#16#0;
   S705_BT_CODE_2013.TEST_TEMP[13] := B#16#0;
   S705_BT_CODE_2013.TEST_TEMP[14] := B#16#0;
   S705_BT_CODE_2013.TEST_TEMP[15] := B#16#0;
   S705_BT_CODE_2013.TEST_TEMP[16] := B#16#0;
   S705_BT_CODE_2013.TEST_TEMP[17] := B#16#0;
   S705_BT_CODE_2013.TEST_TEMP[18] := B#16#0;
   S705_BT_CODE_2013.TEST_TEMP[19] := B#16#0;
   S705_BT_CODE_2013.TEST_TEMP[20] := B#16#0;
   S705_BT_CODE_2013.TEST_TEMP[21] := B#16#0;
   S705_BT_CODE_2013.TEST_TEMP[22] := B#16#0;
   S705_BT_CODE_2013.TEST_TEMP[23] := B#16#0;
   S705_BT_CODE_2013.TEST_TEMP[24] := B#16#0;
   S705_BT_CODE_2013.TEST_TEMP[25] := B#16#0;
   S705_BT_CODE_2013.TEST_TEMP[26] := B#16#0;
   S705_BT_CODE_2013.TEST_TEMP[27] := B#16#0;
   S705_BT_CODE_2013.TEST_TEMP[28] := B#16#0;
   S705_BT_CODE_2013.TEST_TEMP[29] := B#16#0;
   S705_BT_CODE_2013.TEST_TEMP[30] := B#16#0;
   S705_BT_CODE_2013.TEST_TEMP[31] := B#16#0;
   S705_BT_CODE_2013.TEST_TEMP[32] := B#16#0;
   S705_BT_CODE_2013.TEST_TEMP[33] := B#16#0;
   S705_BT_CODE_2013.TEST_TEMP[34] := B#16#0;
   S705_BT_CODE_2013.TEST_TEMP[35] := B#16#0;
   S705_BT_CODE_2013.TEST_TEMP[36] := B#16#0;
   S705_BT_CODE_2013.TEST_TEMP[37] := B#16#0;
   S705_BT_CODE_2013.TEST_TEMP[38] := B#16#0;
   S705_BT_CODE_2013.TEST_TEMP[39] := B#16#0;
   S705_BT_CODE_2013.TEST_TEMP[40] := B#16#0;
   S705_BT_CODE_2014.STATION_MAIN := W#16#0;
   S705_BT_CODE_2014.DISTINCTION_LH_RH := W#16#0;
   S705_BT_CODE_2014.STAION_NUMBER := W#16#0;
   S705_BT_CODE_2014.BODY_TYPE_1ST := W#16#0;
   S705_BT_CODE_2014.BODY_TYPE_OPTION := W#16#0;
   S705_BT_CODE_2014.RBT1_STANDARD_WELD_DATA := W#16#0;
   S705_BT_CODE_2014.RBT2_STANDARD_WELD_DATA := W#16#0;
   S705_BT_CODE_2014.RBT3_STANDARD_WELD_DATA := W#16#0;
   S705_BT_CODE_2014.RBT4_STANDARD_WELD_DATA := W#16#0;
   S705_BT_CODE_2014.RBT5_STANDARD_WELD_DATA := W#16#0;
   S705_BT_CODE_2014.RBT6_STANDARD_WELD_DATA := W#16#0;
   S705_BT_CODE_2014.RBT7_STANDARD_WELD_DATA := W#16#0;
   S705_BT_CODE_2014.RBT8_STANDARD_WELD_DATA := W#16#0;
   S705_BT_CODE_2014.RBT9_STANDARD_WELD_DATA := W#16#0;
   S705_BT_CODE_2014.RBT10_STANDARD_WELD_DATA := W#16#0;
   S705_BT_CODE_2014.RBT11_STANDARD_WELD_DATA := W#16#0;
   S705_BT_CODE_2014.RBT12_STANDARD_WELD_DATA := W#16#0;
   S705_BT_CODE_2014.RBT13_STANDARD_WELD_DATA := W#16#0;
   S705_BT_CODE_2014.RBT14_STANDARD_WELD_DATA := W#16#0;
   S705_BT_CODE_2014.RBT15_STANDARD_WELD_DATA := W#16#0;
   S705_BT_CODE_2014.RBT16_STANDARD_WELD_DATA := W#16#0;
   S705_BT_CODE_2014.RBT17_STANDARD_WELD_DATA := W#16#0;
   S705_BT_CODE_2014.RBT18_STANDARD_WELD_DATA := W#16#0;
   S705_BT_CODE_2014.RBT19_STANDARD_WELD_DATA := W#16#0;
   S705_BT_CODE_2014.RBT20_STANDARD_WELD_DATA := W#16#0;
   S705_BT_CODE_2014.RBT21_STANDARD_WELD_DATA := W#16#0;
   S705_BT_CODE_2014.RBT22_STANDARD_WELD_DATA := W#16#0;
   S705_BT_CODE_2014.RBT23_STANDARD_WELD_DAT := W#16#0;
   S705_BT_CODE_2014.RBT24_STANDARD_WELD_DAT := W#16#0;
   S705_BT_CODE_2014.CHK_WORD := W#16#0;
   S705_BT_CODE_2014.TEST_TEMP[1] := B#16#0;
   S705_BT_CODE_2014.TEST_TEMP[2] := B#16#0;
   S705_BT_CODE_2014.TEST_TEMP[3] := B#16#0;
   S705_BT_CODE_2014.TEST_TEMP[4] := B#16#0;
   S705_BT_CODE_2014.TEST_TEMP[5] := B#16#0;
   S705_BT_CODE_2014.TEST_TEMP[6] := B#16#0;
   S705_BT_CODE_2014.TEST_TEMP[7] := B#16#0;
   S705_BT_CODE_2014.TEST_TEMP[8] := B#16#0;
   S705_BT_CODE_2014.TEST_TEMP[9] := B#16#0;
   S705_BT_CODE_2014.TEST_TEMP[10] := B#16#0;
   S705_BT_CODE_2014.TEST_TEMP[11] := B#16#0;
   S705_BT_CODE_2014.TEST_TEMP[12] := B#16#0;
   S705_BT_CODE_2014.TEST_TEMP[13] := B#16#0;
   S705_BT_CODE_2014.TEST_TEMP[14] := B#16#0;
   S705_BT_CODE_2014.TEST_TEMP[15] := B#16#0;
   S705_BT_CODE_2014.TEST_TEMP[16] := B#16#0;
   S705_BT_CODE_2014.TEST_TEMP[17] := B#16#0;
   S705_BT_CODE_2014.TEST_TEMP[18] := B#16#0;
   S705_BT_CODE_2014.TEST_TEMP[19] := B#16#0;
   S705_BT_CODE_2014.TEST_TEMP[20] := B#16#0;
   S705_BT_CODE_2014.TEST_TEMP[21] := B#16#0;
   S705_BT_CODE_2014.TEST_TEMP[22] := B#16#0;
   S705_BT_CODE_2014.TEST_TEMP[23] := B#16#0;
   S705_BT_CODE_2014.TEST_TEMP[24] := B#16#0;
   S705_BT_CODE_2014.TEST_TEMP[25] := B#16#0;
   S705_BT_CODE_2014.TEST_TEMP[26] := B#16#0;
   S705_BT_CODE_2014.TEST_TEMP[27] := B#16#0;
   S705_BT_CODE_2014.TEST_TEMP[28] := B#16#0;
   S705_BT_CODE_2014.TEST_TEMP[29] := B#16#0;
   S705_BT_CODE_2014.TEST_TEMP[30] := B#16#0;
   S705_BT_CODE_2014.TEST_TEMP[31] := B#16#0;
   S705_BT_CODE_2014.TEST_TEMP[32] := B#16#0;
   S705_BT_CODE_2014.TEST_TEMP[33] := B#16#0;
   S705_BT_CODE_2014.TEST_TEMP[34] := B#16#0;
   S705_BT_CODE_2014.TEST_TEMP[35] := B#16#0;
   S705_BT_CODE_2014.TEST_TEMP[36] := B#16#0;
   S705_BT_CODE_2014.TEST_TEMP[37] := B#16#0;
   S705_BT_CODE_2014.TEST_TEMP[38] := B#16#0;
   S705_BT_CODE_2014.TEST_TEMP[39] := B#16#0;
   S705_BT_CODE_2014.TEST_TEMP[40] := B#16#0;
   S705_BT_CODE_2015.STATION_MAIN := W#16#0;
   S705_BT_CODE_2015.DISTINCTION_LH_RH := W#16#0;
   S705_BT_CODE_2015.STAION_NUMBER := W#16#0;
   S705_BT_CODE_2015.BODY_TYPE_1ST := W#16#0;
   S705_BT_CODE_2015.BODY_TYPE_OPTION := W#16#0;
   S705_BT_CODE_2015.RBT1_STANDARD_WELD_DATA := W#16#0;
   S705_BT_CODE_2015.RBT2_STANDARD_WELD_DATA := W#16#0;
   S705_BT_CODE_2015.RBT3_STANDARD_WELD_DATA := W#16#0;
   S705_BT_CODE_2015.RBT4_STANDARD_WELD_DATA := W#16#0;
   S705_BT_CODE_2015.RBT5_STANDARD_WELD_DATA := W#16#0;
   S705_BT_CODE_2015.RBT6_STANDARD_WELD_DATA := W#16#0;
   S705_BT_CODE_2015.RBT7_STANDARD_WELD_DATA := W#16#0;
   S705_BT_CODE_2015.RBT8_STANDARD_WELD_DATA := W#16#0;
   S705_BT_CODE_2015.RBT9_STANDARD_WELD_DATA := W#16#0;
   S705_BT_CODE_2015.RBT10_STANDARD_WELD_DATA := W#16#0;
   S705_BT_CODE_2015.RBT11_STANDARD_WELD_DATA := W#16#0;
   S705_BT_CODE_2015.RBT12_STANDARD_WELD_DATA := W#16#0;
   S705_BT_CODE_2015.RBT13_STANDARD_WELD_DATA := W#16#0;
   S705_BT_CODE_2015.RBT14_STANDARD_WELD_DATA := W#16#0;
   S705_BT_CODE_2015.RBT15_STANDARD_WELD_DATA := W#16#0;
   S705_BT_CODE_2015.RBT16_STANDARD_WELD_DATA := W#16#0;
   S705_BT_CODE_2015.RBT17_STANDARD_WELD_DATA := W#16#0;
   S705_BT_CODE_2015.RBT18_STANDARD_WELD_DATA := W#16#0;
   S705_BT_CODE_2015.RBT19_STANDARD_WELD_DATA := W#16#0;
   S705_BT_CODE_2015.RBT20_STANDARD_WELD_DATA := W#16#0;
   S705_BT_CODE_2015.RBT21_STANDARD_WELD_DATA := W#16#0;
   S705_BT_CODE_2015.RBT22_STANDARD_WELD_DATA := W#16#0;
   S705_BT_CODE_2015.RBT23_STANDARD_WELD_DAT := W#16#0;
   S705_BT_CODE_2015.RBT24_STANDARD_WELD_DAT := W#16#0;
   S705_BT_CODE_2015.CHK_WORD := W#16#0;
   S705_BT_CODE_2015.TEST_TEMP[1] := B#16#0;
   S705_BT_CODE_2015.TEST_TEMP[2] := B#16#0;
   S705_BT_CODE_2015.TEST_TEMP[3] := B#16#0;
   S705_BT_CODE_2015.TEST_TEMP[4] := B#16#0;
   S705_BT_CODE_2015.TEST_TEMP[5] := B#16#0;
   S705_BT_CODE_2015.TEST_TEMP[6] := B#16#0;
   S705_BT_CODE_2015.TEST_TEMP[7] := B#16#0;
   S705_BT_CODE_2015.TEST_TEMP[8] := B#16#0;
   S705_BT_CODE_2015.TEST_TEMP[9] := B#16#0;
   S705_BT_CODE_2015.TEST_TEMP[10] := B#16#0;
   S705_BT_CODE_2015.TEST_TEMP[11] := B#16#0;
   S705_BT_CODE_2015.TEST_TEMP[12] := B#16#0;
   S705_BT_CODE_2015.TEST_TEMP[13] := B#16#0;
   S705_BT_CODE_2015.TEST_TEMP[14] := B#16#0;
   S705_BT_CODE_2015.TEST_TEMP[15] := B#16#0;
   S705_BT_CODE_2015.TEST_TEMP[16] := B#16#0;
   S705_BT_CODE_2015.TEST_TEMP[17] := B#16#0;
   S705_BT_CODE_2015.TEST_TEMP[18] := B#16#0;
   S705_BT_CODE_2015.TEST_TEMP[19] := B#16#0;
   S705_BT_CODE_2015.TEST_TEMP[20] := B#16#0;
   S705_BT_CODE_2015.TEST_TEMP[21] := B#16#0;
   S705_BT_CODE_2015.TEST_TEMP[22] := B#16#0;
   S705_BT_CODE_2015.TEST_TEMP[23] := B#16#0;
   S705_BT_CODE_2015.TEST_TEMP[24] := B#16#0;
   S705_BT_CODE_2015.TEST_TEMP[25] := B#16#0;
   S705_BT_CODE_2015.TEST_TEMP[26] := B#16#0;
   S705_BT_CODE_2015.TEST_TEMP[27] := B#16#0;
   S705_BT_CODE_2015.TEST_TEMP[28] := B#16#0;
   S705_BT_CODE_2015.TEST_TEMP[29] := B#16#0;
   S705_BT_CODE_2015.TEST_TEMP[30] := B#16#0;
   S705_BT_CODE_2015.TEST_TEMP[31] := B#16#0;
   S705_BT_CODE_2015.TEST_TEMP[32] := B#16#0;
   S705_BT_CODE_2015.TEST_TEMP[33] := B#16#0;
   S705_BT_CODE_2015.TEST_TEMP[34] := B#16#0;
   S705_BT_CODE_2015.TEST_TEMP[35] := B#16#0;
   S705_BT_CODE_2015.TEST_TEMP[36] := B#16#0;
   S705_BT_CODE_2015.TEST_TEMP[37] := B#16#0;
   S705_BT_CODE_2015.TEST_TEMP[38] := B#16#0;
   S705_BT_CODE_2015.TEST_TEMP[39] := B#16#0;
   S705_BT_CODE_2015.TEST_TEMP[40] := B#16#0;
   S705_BT_CODE_2016.STATION_MAIN := W#16#0;
   S705_BT_CODE_2016.DISTINCTION_LH_RH := W#16#0;
   S705_BT_CODE_2016.STAION_NUMBER := W#16#0;
   S705_BT_CODE_2016.BODY_TYPE_1ST := W#16#0;
   S705_BT_CODE_2016.BODY_TYPE_OPTION := W#16#0;
   S705_BT_CODE_2016.RBT1_STANDARD_WELD_DATA := W#16#0;
   S705_BT_CODE_2016.RBT2_STANDARD_WELD_DATA := W#16#0;
   S705_BT_CODE_2016.RBT3_STANDARD_WELD_DATA := W#16#0;
   S705_BT_CODE_2016.RBT4_STANDARD_WELD_DATA := W#16#0;
   S705_BT_CODE_2016.RBT5_STANDARD_WELD_DATA := W#16#0;
   S705_BT_CODE_2016.RBT6_STANDARD_WELD_DATA := W#16#0;
   S705_BT_CODE_2016.RBT7_STANDARD_WELD_DATA := W#16#0;
   S705_BT_CODE_2016.RBT8_STANDARD_WELD_DATA := W#16#0;
   S705_BT_CODE_2016.RBT9_STANDARD_WELD_DATA := W#16#0;
   S705_BT_CODE_2016.RBT10_STANDARD_WELD_DATA := W#16#0;
   S705_BT_CODE_2016.RBT11_STANDARD_WELD_DATA := W#16#0;
   S705_BT_CODE_2016.RBT12_STANDARD_WELD_DATA := W#16#0;
   S705_BT_CODE_2016.RBT13_STANDARD_WELD_DATA := W#16#0;
   S705_BT_CODE_2016.RBT14_STANDARD_WELD_DATA := W#16#0;
   S705_BT_CODE_2016.RBT15_STANDARD_WELD_DATA := W#16#0;
   S705_BT_CODE_2016.RBT16_STANDARD_WELD_DATA := W#16#0;
   S705_BT_CODE_2016.RBT17_STANDARD_WELD_DATA := W#16#0;
   S705_BT_CODE_2016.RBT18_STANDARD_WELD_DATA := W#16#0;
   S705_BT_CODE_2016.RBT19_STANDARD_WELD_DATA := W#16#0;
   S705_BT_CODE_2016.RBT20_STANDARD_WELD_DATA := W#16#0;
   S705_BT_CODE_2016.RBT21_STANDARD_WELD_DATA := W#16#0;
   S705_BT_CODE_2016.RBT22_STANDARD_WELD_DATA := W#16#0;
   S705_BT_CODE_2016.RBT23_STANDARD_WELD_DAT := W#16#0;
   S705_BT_CODE_2016.RBT24_STANDARD_WELD_DAT := W#16#0;
   S705_BT_CODE_2016.CHK_WORD := W#16#0;
   S705_BT_CODE_2016.TEST_TEMP[1] := B#16#0;
   S705_BT_CODE_2016.TEST_TEMP[2] := B#16#0;
   S705_BT_CODE_2016.TEST_TEMP[3] := B#16#0;
   S705_BT_CODE_2016.TEST_TEMP[4] := B#16#0;
   S705_BT_CODE_2016.TEST_TEMP[5] := B#16#0;
   S705_BT_CODE_2016.TEST_TEMP[6] := B#16#0;
   S705_BT_CODE_2016.TEST_TEMP[7] := B#16#0;
   S705_BT_CODE_2016.TEST_TEMP[8] := B#16#0;
   S705_BT_CODE_2016.TEST_TEMP[9] := B#16#0;
   S705_BT_CODE_2016.TEST_TEMP[10] := B#16#0;
   S705_BT_CODE_2016.TEST_TEMP[11] := B#16#0;
   S705_BT_CODE_2016.TEST_TEMP[12] := B#16#0;
   S705_BT_CODE_2016.TEST_TEMP[13] := B#16#0;
   S705_BT_CODE_2016.TEST_TEMP[14] := B#16#0;
   S705_BT_CODE_2016.TEST_TEMP[15] := B#16#0;
   S705_BT_CODE_2016.TEST_TEMP[16] := B#16#0;
   S705_BT_CODE_2016.TEST_TEMP[17] := B#16#0;
   S705_BT_CODE_2016.TEST_TEMP[18] := B#16#0;
   S705_BT_CODE_2016.TEST_TEMP[19] := B#16#0;
   S705_BT_CODE_2016.TEST_TEMP[20] := B#16#0;
   S705_BT_CODE_2016.TEST_TEMP[21] := B#16#0;
   S705_BT_CODE_2016.TEST_TEMP[22] := B#16#0;
   S705_BT_CODE_2016.TEST_TEMP[23] := B#16#0;
   S705_BT_CODE_2016.TEST_TEMP[24] := B#16#0;
   S705_BT_CODE_2016.TEST_TEMP[25] := B#16#0;
   S705_BT_CODE_2016.TEST_TEMP[26] := B#16#0;
   S705_BT_CODE_2016.TEST_TEMP[27] := B#16#0;
   S705_BT_CODE_2016.TEST_TEMP[28] := B#16#0;
   S705_BT_CODE_2016.TEST_TEMP[29] := B#16#0;
   S705_BT_CODE_2016.TEST_TEMP[30] := B#16#0;
   S705_BT_CODE_2016.TEST_TEMP[31] := B#16#0;
   S705_BT_CODE_2016.TEST_TEMP[32] := B#16#0;
   S705_BT_CODE_2016.TEST_TEMP[33] := B#16#0;
   S705_BT_CODE_2016.TEST_TEMP[34] := B#16#0;
   S705_BT_CODE_2016.TEST_TEMP[35] := B#16#0;
   S705_BT_CODE_2016.TEST_TEMP[36] := B#16#0;
   S705_BT_CODE_2016.TEST_TEMP[37] := B#16#0;
   S705_BT_CODE_2016.TEST_TEMP[38] := B#16#0;
   S705_BT_CODE_2016.TEST_TEMP[39] := B#16#0;
   S705_BT_CODE_2016.TEST_TEMP[40] := B#16#0;
   S705_BT_CODE_2017.STATION_MAIN := W#16#0;
   S705_BT_CODE_2017.DISTINCTION_LH_RH := W#16#0;
   S705_BT_CODE_2017.STAION_NUMBER := W#16#0;
   S705_BT_CODE_2017.BODY_TYPE_1ST := W#16#0;
   S705_BT_CODE_2017.BODY_TYPE_OPTION := W#16#0;
   S705_BT_CODE_2017.RBT1_STANDARD_WELD_DATA := W#16#0;
   S705_BT_CODE_2017.RBT2_STANDARD_WELD_DATA := W#16#0;
   S705_BT_CODE_2017.RBT3_STANDARD_WELD_DATA := W#16#0;
   S705_BT_CODE_2017.RBT4_STANDARD_WELD_DATA := W#16#0;
   S705_BT_CODE_2017.RBT5_STANDARD_WELD_DATA := W#16#0;
   S705_BT_CODE_2017.RBT6_STANDARD_WELD_DATA := W#16#0;
   S705_BT_CODE_2017.RBT7_STANDARD_WELD_DATA := W#16#0;
   S705_BT_CODE_2017.RBT8_STANDARD_WELD_DATA := W#16#0;
   S705_BT_CODE_2017.RBT9_STANDARD_WELD_DATA := W#16#0;
   S705_BT_CODE_2017.RBT10_STANDARD_WELD_DATA := W#16#0;
   S705_BT_CODE_2017.RBT11_STANDARD_WELD_DATA := W#16#0;
   S705_BT_CODE_2017.RBT12_STANDARD_WELD_DATA := W#16#0;
   S705_BT_CODE_2017.RBT13_STANDARD_WELD_DATA := W#16#0;
   S705_BT_CODE_2017.RBT14_STANDARD_WELD_DATA := W#16#0;
   S705_BT_CODE_2017.RBT15_STANDARD_WELD_DATA := W#16#0;
   S705_BT_CODE_2017.RBT16_STANDARD_WELD_DATA := W#16#0;
   S705_BT_CODE_2017.RBT17_STANDARD_WELD_DATA := W#16#0;
   S705_BT_CODE_2017.RBT18_STANDARD_WELD_DATA := W#16#0;
   S705_BT_CODE_2017.RBT19_STANDARD_WELD_DATA := W#16#0;
   S705_BT_CODE_2017.RBT20_STANDARD_WELD_DATA := W#16#0;
   S705_BT_CODE_2017.RBT21_STANDARD_WELD_DATA := W#16#0;
   S705_BT_CODE_2017.RBT22_STANDARD_WELD_DATA := W#16#0;
   S705_BT_CODE_2017.RBT23_STANDARD_WELD_DAT := W#16#0;
   S705_BT_CODE_2017.RBT24_STANDARD_WELD_DAT := W#16#0;
   S705_BT_CODE_2017.CHK_WORD := W#16#0;
   S705_BT_CODE_2017.TEST_TEMP[1] := B#16#0;
   S705_BT_CODE_2017.TEST_TEMP[2] := B#16#0;
   S705_BT_CODE_2017.TEST_TEMP[3] := B#16#0;
   S705_BT_CODE_2017.TEST_TEMP[4] := B#16#0;
   S705_BT_CODE_2017.TEST_TEMP[5] := B#16#0;
   S705_BT_CODE_2017.TEST_TEMP[6] := B#16#0;
   S705_BT_CODE_2017.TEST_TEMP[7] := B#16#0;
   S705_BT_CODE_2017.TEST_TEMP[8] := B#16#0;
   S705_BT_CODE_2017.TEST_TEMP[9] := B#16#0;
   S705_BT_CODE_2017.TEST_TEMP[10] := B#16#0;
   S705_BT_CODE_2017.TEST_TEMP[11] := B#16#0;
   S705_BT_CODE_2017.TEST_TEMP[12] := B#16#0;
   S705_BT_CODE_2017.TEST_TEMP[13] := B#16#0;
   S705_BT_CODE_2017.TEST_TEMP[14] := B#16#0;
   S705_BT_CODE_2017.TEST_TEMP[15] := B#16#0;
   S705_BT_CODE_2017.TEST_TEMP[16] := B#16#0;
   S705_BT_CODE_2017.TEST_TEMP[17] := B#16#0;
   S705_BT_CODE_2017.TEST_TEMP[18] := B#16#0;
   S705_BT_CODE_2017.TEST_TEMP[19] := B#16#0;
   S705_BT_CODE_2017.TEST_TEMP[20] := B#16#0;
   S705_BT_CODE_2017.TEST_TEMP[21] := B#16#0;
   S705_BT_CODE_2017.TEST_TEMP[22] := B#16#0;
   S705_BT_CODE_2017.TEST_TEMP[23] := B#16#0;
   S705_BT_CODE_2017.TEST_TEMP[24] := B#16#0;
   S705_BT_CODE_2017.TEST_TEMP[25] := B#16#0;
   S705_BT_CODE_2017.TEST_TEMP[26] := B#16#0;
   S705_BT_CODE_2017.TEST_TEMP[27] := B#16#0;
   S705_BT_CODE_2017.TEST_TEMP[28] := B#16#0;
   S705_BT_CODE_2017.TEST_TEMP[29] := B#16#0;
   S705_BT_CODE_2017.TEST_TEMP[30] := B#16#0;
   S705_BT_CODE_2017.TEST_TEMP[31] := B#16#0;
   S705_BT_CODE_2017.TEST_TEMP[32] := B#16#0;
   S705_BT_CODE_2017.TEST_TEMP[33] := B#16#0;
   S705_BT_CODE_2017.TEST_TEMP[34] := B#16#0;
   S705_BT_CODE_2017.TEST_TEMP[35] := B#16#0;
   S705_BT_CODE_2017.TEST_TEMP[36] := B#16#0;
   S705_BT_CODE_2017.TEST_TEMP[37] := B#16#0;
   S705_BT_CODE_2017.TEST_TEMP[38] := B#16#0;
   S705_BT_CODE_2017.TEST_TEMP[39] := B#16#0;
   S705_BT_CODE_2017.TEST_TEMP[40] := B#16#0;
   S705_BT_CODE_2018.STATION_MAIN := W#16#0;
   S705_BT_CODE_2018.DISTINCTION_LH_RH := W#16#0;
   S705_BT_CODE_2018.STAION_NUMBER := W#16#0;
   S705_BT_CODE_2018.BODY_TYPE_1ST := W#16#0;
   S705_BT_CODE_2018.BODY_TYPE_OPTION := W#16#0;
   S705_BT_CODE_2018.RBT1_STANDARD_WELD_DATA := W#16#0;
   S705_BT_CODE_2018.RBT2_STANDARD_WELD_DATA := W#16#0;
   S705_BT_CODE_2018.RBT3_STANDARD_WELD_DATA := W#16#0;
   S705_BT_CODE_2018.RBT4_STANDARD_WELD_DATA := W#16#0;
   S705_BT_CODE_2018.RBT5_STANDARD_WELD_DATA := W#16#0;
   S705_BT_CODE_2018.RBT6_STANDARD_WELD_DATA := W#16#0;
   S705_BT_CODE_2018.RBT7_STANDARD_WELD_DATA := W#16#0;
   S705_BT_CODE_2018.RBT8_STANDARD_WELD_DATA := W#16#0;
   S705_BT_CODE_2018.RBT9_STANDARD_WELD_DATA := W#16#0;
   S705_BT_CODE_2018.RBT10_STANDARD_WELD_DATA := W#16#0;
   S705_BT_CODE_2018.RBT11_STANDARD_WELD_DATA := W#16#0;
   S705_BT_CODE_2018.RBT12_STANDARD_WELD_DATA := W#16#0;
   S705_BT_CODE_2018.RBT13_STANDARD_WELD_DATA := W#16#0;
   S705_BT_CODE_2018.RBT14_STANDARD_WELD_DATA := W#16#0;
   S705_BT_CODE_2018.RBT15_STANDARD_WELD_DATA := W#16#0;
   S705_BT_CODE_2018.RBT16_STANDARD_WELD_DATA := W#16#0;
   S705_BT_CODE_2018.RBT17_STANDARD_WELD_DATA := W#16#0;
   S705_BT_CODE_2018.RBT18_STANDARD_WELD_DATA := W#16#0;
   S705_BT_CODE_2018.RBT19_STANDARD_WELD_DATA := W#16#0;
   S705_BT_CODE_2018.RBT20_STANDARD_WELD_DATA := W#16#0;
   S705_BT_CODE_2018.RBT21_STANDARD_WELD_DATA := W#16#0;
   S705_BT_CODE_2018.RBT22_STANDARD_WELD_DATA := W#16#0;
   S705_BT_CODE_2018.RBT23_STANDARD_WELD_DAT := W#16#0;
   S705_BT_CODE_2018.RBT24_STANDARD_WELD_DAT := W#16#0;
   S705_BT_CODE_2018.CHK_WORD := W#16#0;
   S705_BT_CODE_2018.TEST_TEMP[1] := B#16#0;
   S705_BT_CODE_2018.TEST_TEMP[2] := B#16#0;
   S705_BT_CODE_2018.TEST_TEMP[3] := B#16#0;
   S705_BT_CODE_2018.TEST_TEMP[4] := B#16#0;
   S705_BT_CODE_2018.TEST_TEMP[5] := B#16#0;
   S705_BT_CODE_2018.TEST_TEMP[6] := B#16#0;
   S705_BT_CODE_2018.TEST_TEMP[7] := B#16#0;
   S705_BT_CODE_2018.TEST_TEMP[8] := B#16#0;
   S705_BT_CODE_2018.TEST_TEMP[9] := B#16#0;
   S705_BT_CODE_2018.TEST_TEMP[10] := B#16#0;
   S705_BT_CODE_2018.TEST_TEMP[11] := B#16#0;
   S705_BT_CODE_2018.TEST_TEMP[12] := B#16#0;
   S705_BT_CODE_2018.TEST_TEMP[13] := B#16#0;
   S705_BT_CODE_2018.TEST_TEMP[14] := B#16#0;
   S705_BT_CODE_2018.TEST_TEMP[15] := B#16#0;
   S705_BT_CODE_2018.TEST_TEMP[16] := B#16#0;
   S705_BT_CODE_2018.TEST_TEMP[17] := B#16#0;
   S705_BT_CODE_2018.TEST_TEMP[18] := B#16#0;
   S705_BT_CODE_2018.TEST_TEMP[19] := B#16#0;
   S705_BT_CODE_2018.TEST_TEMP[20] := B#16#0;
   S705_BT_CODE_2018.TEST_TEMP[21] := B#16#0;
   S705_BT_CODE_2018.TEST_TEMP[22] := B#16#0;
   S705_BT_CODE_2018.TEST_TEMP[23] := B#16#0;
   S705_BT_CODE_2018.TEST_TEMP[24] := B#16#0;
   S705_BT_CODE_2018.TEST_TEMP[25] := B#16#0;
   S705_BT_CODE_2018.TEST_TEMP[26] := B#16#0;
   S705_BT_CODE_2018.TEST_TEMP[27] := B#16#0;
   S705_BT_CODE_2018.TEST_TEMP[28] := B#16#0;
   S705_BT_CODE_2018.TEST_TEMP[29] := B#16#0;
   S705_BT_CODE_2018.TEST_TEMP[30] := B#16#0;
   S705_BT_CODE_2018.TEST_TEMP[31] := B#16#0;
   S705_BT_CODE_2018.TEST_TEMP[32] := B#16#0;
   S705_BT_CODE_2018.TEST_TEMP[33] := B#16#0;
   S705_BT_CODE_2018.TEST_TEMP[34] := B#16#0;
   S705_BT_CODE_2018.TEST_TEMP[35] := B#16#0;
   S705_BT_CODE_2018.TEST_TEMP[36] := B#16#0;
   S705_BT_CODE_2018.TEST_TEMP[37] := B#16#0;
   S705_BT_CODE_2018.TEST_TEMP[38] := B#16#0;
   S705_BT_CODE_2018.TEST_TEMP[39] := B#16#0;
   S705_BT_CODE_2018.TEST_TEMP[40] := B#16#0;
   S705_BT_CODE_2019.STATION_MAIN := W#16#2C1;
   S705_BT_CODE_2019.DISTINCTION_LH_RH := W#16#1;
   S705_BT_CODE_2019.STAION_NUMBER := W#16#0;
   S705_BT_CODE_2019.BODY_TYPE_1ST := W#16#1;
   S705_BT_CODE_2019.BODY_TYPE_OPTION := W#16#7E3;
   S705_BT_CODE_2019.RBT1_STANDARD_WELD_DATA := W#16#3;
   S705_BT_CODE_2019.RBT2_STANDARD_WELD_DATA := W#16#0;
   S705_BT_CODE_2019.RBT3_STANDARD_WELD_DATA := W#16#0;
   S705_BT_CODE_2019.RBT4_STANDARD_WELD_DATA := W#16#0;
   S705_BT_CODE_2019.RBT5_STANDARD_WELD_DATA := W#16#0;
   S705_BT_CODE_2019.RBT6_STANDARD_WELD_DATA := W#16#0;
   S705_BT_CODE_2019.RBT7_STANDARD_WELD_DATA := W#16#0;
   S705_BT_CODE_2019.RBT8_STANDARD_WELD_DATA := W#16#0;
   S705_BT_CODE_2019.RBT9_STANDARD_WELD_DATA := W#16#0;
   S705_BT_CODE_2019.RBT10_STANDARD_WELD_DATA := W#16#0;
   S705_BT_CODE_2019.RBT11_STANDARD_WELD_DATA := W#16#0;
   S705_BT_CODE_2019.RBT12_STANDARD_WELD_DATA := W#16#0;
   S705_BT_CODE_2019.RBT13_STANDARD_WELD_DATA := W#16#0;
   S705_BT_CODE_2019.RBT14_STANDARD_WELD_DATA := W#16#0;
   S705_BT_CODE_2019.RBT15_STANDARD_WELD_DATA := W#16#0;
   S705_BT_CODE_2019.RBT16_STANDARD_WELD_DATA := W#16#0;
   S705_BT_CODE_2019.RBT17_STANDARD_WELD_DATA := W#16#0;
   S705_BT_CODE_2019.RBT18_STANDARD_WELD_DATA := W#16#0;
   S705_BT_CODE_2019.RBT19_STANDARD_WELD_DATA := W#16#0;
   S705_BT_CODE_2019.RBT20_STANDARD_WELD_DATA := W#16#0;
   S705_BT_CODE_2019.RBT21_STANDARD_WELD_DATA := W#16#0;
   S705_BT_CODE_2019.RBT22_STANDARD_WELD_DATA := W#16#0;
   S705_BT_CODE_2019.RBT23_STANDARD_WELD_DAT := W#16#0;
   S705_BT_CODE_2019.RBT24_STANDARD_WELD_DAT := W#16#0;
   S705_BT_CODE_2019.CHK_WORD := W#16#0;
   S705_BT_CODE_2019.TEST_TEMP[1] := B#16#0;
   S705_BT_CODE_2019.TEST_TEMP[2] := B#16#0;
   S705_BT_CODE_2019.TEST_TEMP[3] := B#16#0;
   S705_BT_CODE_2019.TEST_TEMP[4] := B#16#0;
   S705_BT_CODE_2019.TEST_TEMP[5] := B#16#0;
   S705_BT_CODE_2019.TEST_TEMP[6] := B#16#0;
   S705_BT_CODE_2019.TEST_TEMP[7] := B#16#0;
   S705_BT_CODE_2019.TEST_TEMP[8] := B#16#0;
   S705_BT_CODE_2019.TEST_TEMP[9] := B#16#0;
   S705_BT_CODE_2019.TEST_TEMP[10] := B#16#0;
   S705_BT_CODE_2019.TEST_TEMP[11] := B#16#0;
   S705_BT_CODE_2019.TEST_TEMP[12] := B#16#0;
   S705_BT_CODE_2019.TEST_TEMP[13] := B#16#0;
   S705_BT_CODE_2019.TEST_TEMP[14] := B#16#0;
   S705_BT_CODE_2019.TEST_TEMP[15] := B#16#0;
   S705_BT_CODE_2019.TEST_TEMP[16] := B#16#0;
   S705_BT_CODE_2019.TEST_TEMP[17] := B#16#0;
   S705_BT_CODE_2019.TEST_TEMP[18] := B#16#0;
   S705_BT_CODE_2019.TEST_TEMP[19] := B#16#0;
   S705_BT_CODE_2019.TEST_TEMP[20] := B#16#0;
   S705_BT_CODE_2019.TEST_TEMP[21] := B#16#0;
   S705_BT_CODE_2019.TEST_TEMP[22] := B#16#0;
   S705_BT_CODE_2019.TEST_TEMP[23] := B#16#0;
   S705_BT_CODE_2019.TEST_TEMP[24] := B#16#0;
   S705_BT_CODE_2019.TEST_TEMP[25] := B#16#0;
   S705_BT_CODE_2019.TEST_TEMP[26] := B#16#0;
   S705_BT_CODE_2019.TEST_TEMP[27] := B#16#0;
   S705_BT_CODE_2019.TEST_TEMP[28] := B#16#0;
   S705_BT_CODE_2019.TEST_TEMP[29] := B#16#0;
   S705_BT_CODE_2019.TEST_TEMP[30] := B#16#0;
   S705_BT_CODE_2019.TEST_TEMP[31] := B#16#0;
   S705_BT_CODE_2019.TEST_TEMP[32] := B#16#0;
   S705_BT_CODE_2019.TEST_TEMP[33] := B#16#0;
   S705_BT_CODE_2019.TEST_TEMP[34] := B#16#0;
   S705_BT_CODE_2019.TEST_TEMP[35] := B#16#0;
   S705_BT_CODE_2019.TEST_TEMP[36] := B#16#0;
   S705_BT_CODE_2019.TEST_TEMP[37] := B#16#0;
   S705_BT_CODE_2019.TEST_TEMP[38] := B#16#0;
   S705_BT_CODE_2019.TEST_TEMP[39] := B#16#0;
   S705_BT_CODE_2019.TEST_TEMP[40] := B#16#0;
   S705_BT_CODE_2020.STATION_MAIN := W#16#0;
   S705_BT_CODE_2020.DISTINCTION_LH_RH := W#16#0;
   S705_BT_CODE_2020.STAION_NUMBER := W#16#0;
   S705_BT_CODE_2020.BODY_TYPE_1ST := W#16#0;
   S705_BT_CODE_2020.BODY_TYPE_OPTION := W#16#0;
   S705_BT_CODE_2020.RBT1_STANDARD_WELD_DATA := W#16#0;
   S705_BT_CODE_2020.RBT2_STANDARD_WELD_DATA := W#16#0;
   S705_BT_CODE_2020.RBT3_STANDARD_WELD_DATA := W#16#0;
   S705_BT_CODE_2020.RBT4_STANDARD_WELD_DATA := W#16#0;
   S705_BT_CODE_2020.RBT5_STANDARD_WELD_DATA := W#16#0;
   S705_BT_CODE_2020.RBT6_STANDARD_WELD_DATA := W#16#0;
   S705_BT_CODE_2020.RBT7_STANDARD_WELD_DATA := W#16#0;
   S705_BT_CODE_2020.RBT8_STANDARD_WELD_DATA := W#16#0;
   S705_BT_CODE_2020.RBT9_STANDARD_WELD_DATA := W#16#0;
   S705_BT_CODE_2020.RBT10_STANDARD_WELD_DATA := W#16#0;
   S705_BT_CODE_2020.RBT11_STANDARD_WELD_DATA := W#16#0;
   S705_BT_CODE_2020.RBT12_STANDARD_WELD_DATA := W#16#0;
   S705_BT_CODE_2020.RBT13_STANDARD_WELD_DATA := W#16#0;
   S705_BT_CODE_2020.RBT14_STANDARD_WELD_DATA := W#16#0;
   S705_BT_CODE_2020.RBT15_STANDARD_WELD_DATA := W#16#0;
   S705_BT_CODE_2020.RBT16_STANDARD_WELD_DATA := W#16#0;
   S705_BT_CODE_2020.RBT17_STANDARD_WELD_DATA := W#16#0;
   S705_BT_CODE_2020.RBT18_STANDARD_WELD_DATA := W#16#0;
   S705_BT_CODE_2020.RBT19_STANDARD_WELD_DATA := W#16#0;
   S705_BT_CODE_2020.RBT20_STANDARD_WELD_DATA := W#16#0;
   S705_BT_CODE_2020.RBT21_STANDARD_WELD_DATA := W#16#0;
   S705_BT_CODE_2020.RBT22_STANDARD_WELD_DATA := W#16#0;
   S705_BT_CODE_2020.RBT23_STANDARD_WELD_DAT := W#16#0;
   S705_BT_CODE_2020.RBT24_STANDARD_WELD_DAT := W#16#0;
   S705_BT_CODE_2020.CHK_WORD := W#16#0;
   S705_BT_CODE_2020.TEST_TEMP[1] := B#16#0;
   S705_BT_CODE_2020.TEST_TEMP[2] := B#16#0;
   S705_BT_CODE_2020.TEST_TEMP[3] := B#16#0;
   S705_BT_CODE_2020.TEST_TEMP[4] := B#16#0;
   S705_BT_CODE_2020.TEST_TEMP[5] := B#16#0;
   S705_BT_CODE_2020.TEST_TEMP[6] := B#16#0;
   S705_BT_CODE_2020.TEST_TEMP[7] := B#16#0;
   S705_BT_CODE_2020.TEST_TEMP[8] := B#16#0;
   S705_BT_CODE_2020.TEST_TEMP[9] := B#16#0;
   S705_BT_CODE_2020.TEST_TEMP[10] := B#16#0;
   S705_BT_CODE_2020.TEST_TEMP[11] := B#16#0;
   S705_BT_CODE_2020.TEST_TEMP[12] := B#16#0;
   S705_BT_CODE_2020.TEST_TEMP[13] := B#16#0;
   S705_BT_CODE_2020.TEST_TEMP[14] := B#16#0;
   S705_BT_CODE_2020.TEST_TEMP[15] := B#16#0;
   S705_BT_CODE_2020.TEST_TEMP[16] := B#16#0;
   S705_BT_CODE_2020.TEST_TEMP[17] := B#16#0;
   S705_BT_CODE_2020.TEST_TEMP[18] := B#16#0;
   S705_BT_CODE_2020.TEST_TEMP[19] := B#16#0;
   S705_BT_CODE_2020.TEST_TEMP[20] := B#16#0;
   S705_BT_CODE_2020.TEST_TEMP[21] := B#16#0;
   S705_BT_CODE_2020.TEST_TEMP[22] := B#16#0;
   S705_BT_CODE_2020.TEST_TEMP[23] := B#16#0;
   S705_BT_CODE_2020.TEST_TEMP[24] := B#16#0;
   S705_BT_CODE_2020.TEST_TEMP[25] := B#16#0;
   S705_BT_CODE_2020.TEST_TEMP[26] := B#16#0;
   S705_BT_CODE_2020.TEST_TEMP[27] := B#16#0;
   S705_BT_CODE_2020.TEST_TEMP[28] := B#16#0;
   S705_BT_CODE_2020.TEST_TEMP[29] := B#16#0;
   S705_BT_CODE_2020.TEST_TEMP[30] := B#16#0;
   S705_BT_CODE_2020.TEST_TEMP[31] := B#16#0;
   S705_BT_CODE_2020.TEST_TEMP[32] := B#16#0;
   S705_BT_CODE_2020.TEST_TEMP[33] := B#16#0;
   S705_BT_CODE_2020.TEST_TEMP[34] := B#16#0;
   S705_BT_CODE_2020.TEST_TEMP[35] := B#16#0;
   S705_BT_CODE_2020.TEST_TEMP[36] := B#16#0;
   S705_BT_CODE_2020.TEST_TEMP[37] := B#16#0;
   S705_BT_CODE_2020.TEST_TEMP[38] := B#16#0;
   S705_BT_CODE_2020.TEST_TEMP[39] := B#16#0;
   S705_BT_CODE_2020.TEST_TEMP[40] := B#16#0;
   S705_BT_CODE_2021.STATION_MAIN := W#16#0;
   S705_BT_CODE_2021.DISTINCTION_LH_RH := W#16#0;
   S705_BT_CODE_2021.STAION_NUMBER := W#16#0;
   S705_BT_CODE_2021.BODY_TYPE_1ST := W#16#0;
   S705_BT_CODE_2021.BODY_TYPE_OPTION := W#16#0;
   S705_BT_CODE_2021.RBT1_STANDARD_WELD_DATA := W#16#0;
   S705_BT_CODE_2021.RBT2_STANDARD_WELD_DATA := W#16#0;
   S705_BT_CODE_2021.RBT3_STANDARD_WELD_DATA := W#16#0;
   S705_BT_CODE_2021.RBT4_STANDARD_WELD_DATA := W#16#0;
   S705_BT_CODE_2021.RBT5_STANDARD_WELD_DATA := W#16#0;
   S705_BT_CODE_2021.RBT6_STANDARD_WELD_DATA := W#16#0;
   S705_BT_CODE_2021.RBT7_STANDARD_WELD_DATA := W#16#0;
   S705_BT_CODE_2021.RBT8_STANDARD_WELD_DATA := W#16#0;
   S705_BT_CODE_2021.RBT9_STANDARD_WELD_DATA := W#16#0;
   S705_BT_CODE_2021.RBT10_STANDARD_WELD_DATA := W#16#0;
   S705_BT_CODE_2021.RBT11_STANDARD_WELD_DATA := W#16#0;
   S705_BT_CODE_2021.RBT12_STANDARD_WELD_DATA := W#16#0;
   S705_BT_CODE_2021.RBT13_STANDARD_WELD_DATA := W#16#0;
   S705_BT_CODE_2021.RBT14_STANDARD_WELD_DATA := W#16#0;
   S705_BT_CODE_2021.RBT15_STANDARD_WELD_DATA := W#16#0;
   S705_BT_CODE_2021.RBT16_STANDARD_WELD_DATA := W#16#0;
   S705_BT_CODE_2021.RBT17_STANDARD_WELD_DATA := W#16#0;
   S705_BT_CODE_2021.RBT18_STANDARD_WELD_DATA := W#16#0;
   S705_BT_CODE_2021.RBT19_STANDARD_WELD_DATA := W#16#0;
   S705_BT_CODE_2021.RBT20_STANDARD_WELD_DATA := W#16#0;
   S705_BT_CODE_2021.RBT21_STANDARD_WELD_DATA := W#16#0;
   S705_BT_CODE_2021.RBT22_STANDARD_WELD_DATA := W#16#0;
   S705_BT_CODE_2021.RBT23_STANDARD_WELD_DAT := W#16#0;
   S705_BT_CODE_2021.RBT24_STANDARD_WELD_DAT := W#16#0;
   S705_BT_CODE_2021.CHK_WORD := W#16#0;
   S705_BT_CODE_2021.TEST_TEMP[1] := B#16#0;
   S705_BT_CODE_2021.TEST_TEMP[2] := B#16#0;
   S705_BT_CODE_2021.TEST_TEMP[3] := B#16#0;
   S705_BT_CODE_2021.TEST_TEMP[4] := B#16#0;
   S705_BT_CODE_2021.TEST_TEMP[5] := B#16#0;
   S705_BT_CODE_2021.TEST_TEMP[6] := B#16#0;
   S705_BT_CODE_2021.TEST_TEMP[7] := B#16#0;
   S705_BT_CODE_2021.TEST_TEMP[8] := B#16#0;
   S705_BT_CODE_2021.TEST_TEMP[9] := B#16#0;
   S705_BT_CODE_2021.TEST_TEMP[10] := B#16#0;
   S705_BT_CODE_2021.TEST_TEMP[11] := B#16#0;
   S705_BT_CODE_2021.TEST_TEMP[12] := B#16#0;
   S705_BT_CODE_2021.TEST_TEMP[13] := B#16#0;
   S705_BT_CODE_2021.TEST_TEMP[14] := B#16#0;
   S705_BT_CODE_2021.TEST_TEMP[15] := B#16#0;
   S705_BT_CODE_2021.TEST_TEMP[16] := B#16#0;
   S705_BT_CODE_2021.TEST_TEMP[17] := B#16#0;
   S705_BT_CODE_2021.TEST_TEMP[18] := B#16#0;
   S705_BT_CODE_2021.TEST_TEMP[19] := B#16#0;
   S705_BT_CODE_2021.TEST_TEMP[20] := B#16#0;
   S705_BT_CODE_2021.TEST_TEMP[21] := B#16#0;
   S705_BT_CODE_2021.TEST_TEMP[22] := B#16#0;
   S705_BT_CODE_2021.TEST_TEMP[23] := B#16#0;
   S705_BT_CODE_2021.TEST_TEMP[24] := B#16#0;
   S705_BT_CODE_2021.TEST_TEMP[25] := B#16#0;
   S705_BT_CODE_2021.TEST_TEMP[26] := B#16#0;
   S705_BT_CODE_2021.TEST_TEMP[27] := B#16#0;
   S705_BT_CODE_2021.TEST_TEMP[28] := B#16#0;
   S705_BT_CODE_2021.TEST_TEMP[29] := B#16#0;
   S705_BT_CODE_2021.TEST_TEMP[30] := B#16#0;
   S705_BT_CODE_2021.TEST_TEMP[31] := B#16#0;
   S705_BT_CODE_2021.TEST_TEMP[32] := B#16#0;
   S705_BT_CODE_2021.TEST_TEMP[33] := B#16#0;
   S705_BT_CODE_2021.TEST_TEMP[34] := B#16#0;
   S705_BT_CODE_2021.TEST_TEMP[35] := B#16#0;
   S705_BT_CODE_2021.TEST_TEMP[36] := B#16#0;
   S705_BT_CODE_2021.TEST_TEMP[37] := B#16#0;
   S705_BT_CODE_2021.TEST_TEMP[38] := B#16#0;
   S705_BT_CODE_2021.TEST_TEMP[39] := B#16#0;
   S705_BT_CODE_2021.TEST_TEMP[40] := B#16#0;
   S705_BT_CODE_2022.STATION_MAIN := W#16#0;
   S705_BT_CODE_2022.DISTINCTION_LH_RH := W#16#0;
   S705_BT_CODE_2022.STAION_NUMBER := W#16#0;
   S705_BT_CODE_2022.BODY_TYPE_1ST := W#16#0;
   S705_BT_CODE_2022.BODY_TYPE_OPTION := W#16#0;
   S705_BT_CODE_2022.RBT1_STANDARD_WELD_DATA := W#16#0;
   S705_BT_CODE_2022.RBT2_STANDARD_WELD_DATA := W#16#0;
   S705_BT_CODE_2022.RBT3_STANDARD_WELD_DATA := W#16#0;
   S705_BT_CODE_2022.RBT4_STANDARD_WELD_DATA := W#16#0;
   S705_BT_CODE_2022.RBT5_STANDARD_WELD_DATA := W#16#0;
   S705_BT_CODE_2022.RBT6_STANDARD_WELD_DATA := W#16#0;
   S705_BT_CODE_2022.RBT7_STANDARD_WELD_DATA := W#16#0;
   S705_BT_CODE_2022.RBT8_STANDARD_WELD_DATA := W#16#0;
   S705_BT_CODE_2022.RBT9_STANDARD_WELD_DATA := W#16#0;
   S705_BT_CODE_2022.RBT10_STANDARD_WELD_DATA := W#16#0;
   S705_BT_CODE_2022.RBT11_STANDARD_WELD_DATA := W#16#0;
   S705_BT_CODE_2022.RBT12_STANDARD_WELD_DATA := W#16#0;
   S705_BT_CODE_2022.RBT13_STANDARD_WELD_DATA := W#16#0;
   S705_BT_CODE_2022.RBT14_STANDARD_WELD_DATA := W#16#0;
   S705_BT_CODE_2022.RBT15_STANDARD_WELD_DATA := W#16#0;
   S705_BT_CODE_2022.RBT16_STANDARD_WELD_DATA := W#16#0;
   S705_BT_CODE_2022.RBT17_STANDARD_WELD_DATA := W#16#0;
   S705_BT_CODE_2022.RBT18_STANDARD_WELD_DATA := W#16#0;
   S705_BT_CODE_2022.RBT19_STANDARD_WELD_DATA := W#16#0;
   S705_BT_CODE_2022.RBT20_STANDARD_WELD_DATA := W#16#0;
   S705_BT_CODE_2022.RBT21_STANDARD_WELD_DATA := W#16#0;
   S705_BT_CODE_2022.RBT22_STANDARD_WELD_DATA := W#16#0;
   S705_BT_CODE_2022.RBT23_STANDARD_WELD_DAT := W#16#0;
   S705_BT_CODE_2022.RBT24_STANDARD_WELD_DAT := W#16#0;
   S705_BT_CODE_2022.CHK_WORD := W#16#0;
   S705_BT_CODE_2022.TEST_TEMP[1] := B#16#0;
   S705_BT_CODE_2022.TEST_TEMP[2] := B#16#0;
   S705_BT_CODE_2022.TEST_TEMP[3] := B#16#0;
   S705_BT_CODE_2022.TEST_TEMP[4] := B#16#0;
   S705_BT_CODE_2022.TEST_TEMP[5] := B#16#0;
   S705_BT_CODE_2022.TEST_TEMP[6] := B#16#0;
   S705_BT_CODE_2022.TEST_TEMP[7] := B#16#0;
   S705_BT_CODE_2022.TEST_TEMP[8] := B#16#0;
   S705_BT_CODE_2022.TEST_TEMP[9] := B#16#0;
   S705_BT_CODE_2022.TEST_TEMP[10] := B#16#0;
   S705_BT_CODE_2022.TEST_TEMP[11] := B#16#0;
   S705_BT_CODE_2022.TEST_TEMP[12] := B#16#0;
   S705_BT_CODE_2022.TEST_TEMP[13] := B#16#0;
   S705_BT_CODE_2022.TEST_TEMP[14] := B#16#0;
   S705_BT_CODE_2022.TEST_TEMP[15] := B#16#0;
   S705_BT_CODE_2022.TEST_TEMP[16] := B#16#0;
   S705_BT_CODE_2022.TEST_TEMP[17] := B#16#0;
   S705_BT_CODE_2022.TEST_TEMP[18] := B#16#0;
   S705_BT_CODE_2022.TEST_TEMP[19] := B#16#0;
   S705_BT_CODE_2022.TEST_TEMP[20] := B#16#0;
   S705_BT_CODE_2022.TEST_TEMP[21] := B#16#0;
   S705_BT_CODE_2022.TEST_TEMP[22] := B#16#0;
   S705_BT_CODE_2022.TEST_TEMP[23] := B#16#0;
   S705_BT_CODE_2022.TEST_TEMP[24] := B#16#0;
   S705_BT_CODE_2022.TEST_TEMP[25] := B#16#0;
   S705_BT_CODE_2022.TEST_TEMP[26] := B#16#0;
   S705_BT_CODE_2022.TEST_TEMP[27] := B#16#0;
   S705_BT_CODE_2022.TEST_TEMP[28] := B#16#0;
   S705_BT_CODE_2022.TEST_TEMP[29] := B#16#0;
   S705_BT_CODE_2022.TEST_TEMP[30] := B#16#0;
   S705_BT_CODE_2022.TEST_TEMP[31] := B#16#0;
   S705_BT_CODE_2022.TEST_TEMP[32] := B#16#0;
   S705_BT_CODE_2022.TEST_TEMP[33] := B#16#0;
   S705_BT_CODE_2022.TEST_TEMP[34] := B#16#0;
   S705_BT_CODE_2022.TEST_TEMP[35] := B#16#0;
   S705_BT_CODE_2022.TEST_TEMP[36] := B#16#0;
   S705_BT_CODE_2022.TEST_TEMP[37] := B#16#0;
   S705_BT_CODE_2022.TEST_TEMP[38] := B#16#0;
   S705_BT_CODE_2022.TEST_TEMP[39] := B#16#0;
   S705_BT_CODE_2022.TEST_TEMP[40] := B#16#0;
   S705_BT_CODE_2023.STATION_MAIN := W#16#0;
   S705_BT_CODE_2023.DISTINCTION_LH_RH := W#16#0;
   S705_BT_CODE_2023.STAION_NUMBER := W#16#0;
   S705_BT_CODE_2023.BODY_TYPE_1ST := W#16#0;
   S705_BT_CODE_2023.BODY_TYPE_OPTION := W#16#0;
   S705_BT_CODE_2023.RBT1_STANDARD_WELD_DATA := W#16#0;
   S705_BT_CODE_2023.RBT2_STANDARD_WELD_DATA := W#16#0;
   S705_BT_CODE_2023.RBT3_STANDARD_WELD_DATA := W#16#0;
   S705_BT_CODE_2023.RBT4_STANDARD_WELD_DATA := W#16#0;
   S705_BT_CODE_2023.RBT5_STANDARD_WELD_DATA := W#16#0;
   S705_BT_CODE_2023.RBT6_STANDARD_WELD_DATA := W#16#0;
   S705_BT_CODE_2023.RBT7_STANDARD_WELD_DATA := W#16#0;
   S705_BT_CODE_2023.RBT8_STANDARD_WELD_DATA := W#16#0;
   S705_BT_CODE_2023.RBT9_STANDARD_WELD_DATA := W#16#0;
   S705_BT_CODE_2023.RBT10_STANDARD_WELD_DATA := W#16#0;
   S705_BT_CODE_2023.RBT11_STANDARD_WELD_DATA := W#16#0;
   S705_BT_CODE_2023.RBT12_STANDARD_WELD_DATA := W#16#0;
   S705_BT_CODE_2023.RBT13_STANDARD_WELD_DATA := W#16#0;
   S705_BT_CODE_2023.RBT14_STANDARD_WELD_DATA := W#16#0;
   S705_BT_CODE_2023.RBT15_STANDARD_WELD_DATA := W#16#0;
   S705_BT_CODE_2023.RBT16_STANDARD_WELD_DATA := W#16#0;
   S705_BT_CODE_2023.RBT17_STANDARD_WELD_DATA := W#16#0;
   S705_BT_CODE_2023.RBT18_STANDARD_WELD_DATA := W#16#0;
   S705_BT_CODE_2023.RBT19_STANDARD_WELD_DATA := W#16#0;
   S705_BT_CODE_2023.RBT20_STANDARD_WELD_DATA := W#16#0;
   S705_BT_CODE_2023.RBT21_STANDARD_WELD_DATA := W#16#0;
   S705_BT_CODE_2023.RBT22_STANDARD_WELD_DATA := W#16#0;
   S705_BT_CODE_2023.RBT23_STANDARD_WELD_DAT := W#16#0;
   S705_BT_CODE_2023.RBT24_STANDARD_WELD_DAT := W#16#0;
   S705_BT_CODE_2023.CHK_WORD := W#16#0;
   S705_BT_CODE_2023.TEST_TEMP[1] := B#16#0;
   S705_BT_CODE_2023.TEST_TEMP[2] := B#16#0;
   S705_BT_CODE_2023.TEST_TEMP[3] := B#16#0;
   S705_BT_CODE_2023.TEST_TEMP[4] := B#16#0;
   S705_BT_CODE_2023.TEST_TEMP[5] := B#16#0;
   S705_BT_CODE_2023.TEST_TEMP[6] := B#16#0;
   S705_BT_CODE_2023.TEST_TEMP[7] := B#16#0;
   S705_BT_CODE_2023.TEST_TEMP[8] := B#16#0;
   S705_BT_CODE_2023.TEST_TEMP[9] := B#16#0;
   S705_BT_CODE_2023.TEST_TEMP[10] := B#16#0;
   S705_BT_CODE_2023.TEST_TEMP[11] := B#16#0;
   S705_BT_CODE_2023.TEST_TEMP[12] := B#16#0;
   S705_BT_CODE_2023.TEST_TEMP[13] := B#16#0;
   S705_BT_CODE_2023.TEST_TEMP[14] := B#16#0;
   S705_BT_CODE_2023.TEST_TEMP[15] := B#16#0;
   S705_BT_CODE_2023.TEST_TEMP[16] := B#16#0;
   S705_BT_CODE_2023.TEST_TEMP[17] := B#16#0;
   S705_BT_CODE_2023.TEST_TEMP[18] := B#16#0;
   S705_BT_CODE_2023.TEST_TEMP[19] := B#16#0;
   S705_BT_CODE_2023.TEST_TEMP[20] := B#16#0;
   S705_BT_CODE_2023.TEST_TEMP[21] := B#16#0;
   S705_BT_CODE_2023.TEST_TEMP[22] := B#16#0;
   S705_BT_CODE_2023.TEST_TEMP[23] := B#16#0;
   S705_BT_CODE_2023.TEST_TEMP[24] := B#16#0;
   S705_BT_CODE_2023.TEST_TEMP[25] := B#16#0;
   S705_BT_CODE_2023.TEST_TEMP[26] := B#16#0;
   S705_BT_CODE_2023.TEST_TEMP[27] := B#16#0;
   S705_BT_CODE_2023.TEST_TEMP[28] := B#16#0;
   S705_BT_CODE_2023.TEST_TEMP[29] := B#16#0;
   S705_BT_CODE_2023.TEST_TEMP[30] := B#16#0;
   S705_BT_CODE_2023.TEST_TEMP[31] := B#16#0;
   S705_BT_CODE_2023.TEST_TEMP[32] := B#16#0;
   S705_BT_CODE_2023.TEST_TEMP[33] := B#16#0;
   S705_BT_CODE_2023.TEST_TEMP[34] := B#16#0;
   S705_BT_CODE_2023.TEST_TEMP[35] := B#16#0;
   S705_BT_CODE_2023.TEST_TEMP[36] := B#16#0;
   S705_BT_CODE_2023.TEST_TEMP[37] := B#16#0;
   S705_BT_CODE_2023.TEST_TEMP[38] := B#16#0;
   S705_BT_CODE_2023.TEST_TEMP[39] := B#16#0;
   S705_BT_CODE_2023.TEST_TEMP[40] := B#16#0;
   S705_BT_CODE_2024.STATION_MAIN := W#16#0;
   S705_BT_CODE_2024.DISTINCTION_LH_RH := W#16#0;
   S705_BT_CODE_2024.STAION_NUMBER := W#16#0;
   S705_BT_CODE_2024.BODY_TYPE_1ST := W#16#0;
   S705_BT_CODE_2024.BODY_TYPE_OPTION := W#16#0;
   S705_BT_CODE_2024.RBT1_STANDARD_WELD_DATA := W#16#0;
   S705_BT_CODE_2024.RBT2_STANDARD_WELD_DATA := W#16#0;
   S705_BT_CODE_2024.RBT3_STANDARD_WELD_DATA := W#16#0;
   S705_BT_CODE_2024.RBT4_STANDARD_WELD_DATA := W#16#0;
   S705_BT_CODE_2024.RBT5_STANDARD_WELD_DATA := W#16#0;
   S705_BT_CODE_2024.RBT6_STANDARD_WELD_DATA := W#16#0;
   S705_BT_CODE_2024.RBT7_STANDARD_WELD_DATA := W#16#0;
   S705_BT_CODE_2024.RBT8_STANDARD_WELD_DATA := W#16#0;
   S705_BT_CODE_2024.RBT9_STANDARD_WELD_DATA := W#16#0;
   S705_BT_CODE_2024.RBT10_STANDARD_WELD_DATA := W#16#0;
   S705_BT_CODE_2024.RBT11_STANDARD_WELD_DATA := W#16#0;
   S705_BT_CODE_2024.RBT12_STANDARD_WELD_DATA := W#16#0;
   S705_BT_CODE_2024.RBT13_STANDARD_WELD_DATA := W#16#0;
   S705_BT_CODE_2024.RBT14_STANDARD_WELD_DATA := W#16#0;
   S705_BT_CODE_2024.RBT15_STANDARD_WELD_DATA := W#16#0;
   S705_BT_CODE_2024.RBT16_STANDARD_WELD_DATA := W#16#0;
   S705_BT_CODE_2024.RBT17_STANDARD_WELD_DATA := W#16#0;
   S705_BT_CODE_2024.RBT18_STANDARD_WELD_DATA := W#16#0;
   S705_BT_CODE_2024.RBT19_STANDARD_WELD_DATA := W#16#0;
   S705_BT_CODE_2024.RBT20_STANDARD_WELD_DATA := W#16#0;
   S705_BT_CODE_2024.RBT21_STANDARD_WELD_DATA := W#16#0;
   S705_BT_CODE_2024.RBT22_STANDARD_WELD_DATA := W#16#0;
   S705_BT_CODE_2024.RBT23_STANDARD_WELD_DAT := W#16#0;
   S705_BT_CODE_2024.RBT24_STANDARD_WELD_DAT := W#16#0;
   S705_BT_CODE_2024.CHK_WORD := W#16#0;
   S705_BT_CODE_2024.TEST_TEMP[1] := B#16#0;
   S705_BT_CODE_2024.TEST_TEMP[2] := B#16#0;
   S705_BT_CODE_2024.TEST_TEMP[3] := B#16#0;
   S705_BT_CODE_2024.TEST_TEMP[4] := B#16#0;
   S705_BT_CODE_2024.TEST_TEMP[5] := B#16#0;
   S705_BT_CODE_2024.TEST_TEMP[6] := B#16#0;
   S705_BT_CODE_2024.TEST_TEMP[7] := B#16#0;
   S705_BT_CODE_2024.TEST_TEMP[8] := B#16#0;
   S705_BT_CODE_2024.TEST_TEMP[9] := B#16#0;
   S705_BT_CODE_2024.TEST_TEMP[10] := B#16#0;
   S705_BT_CODE_2024.TEST_TEMP[11] := B#16#0;
   S705_BT_CODE_2024.TEST_TEMP[12] := B#16#0;
   S705_BT_CODE_2024.TEST_TEMP[13] := B#16#0;
   S705_BT_CODE_2024.TEST_TEMP[14] := B#16#0;
   S705_BT_CODE_2024.TEST_TEMP[15] := B#16#0;
   S705_BT_CODE_2024.TEST_TEMP[16] := B#16#0;
   S705_BT_CODE_2024.TEST_TEMP[17] := B#16#0;
   S705_BT_CODE_2024.TEST_TEMP[18] := B#16#0;
   S705_BT_CODE_2024.TEST_TEMP[19] := B#16#0;
   S705_BT_CODE_2024.TEST_TEMP[20] := B#16#0;
   S705_BT_CODE_2024.TEST_TEMP[21] := B#16#0;
   S705_BT_CODE_2024.TEST_TEMP[22] := B#16#0;
   S705_BT_CODE_2024.TEST_TEMP[23] := B#16#0;
   S705_BT_CODE_2024.TEST_TEMP[24] := B#16#0;
   S705_BT_CODE_2024.TEST_TEMP[25] := B#16#0;
   S705_BT_CODE_2024.TEST_TEMP[26] := B#16#0;
   S705_BT_CODE_2024.TEST_TEMP[27] := B#16#0;
   S705_BT_CODE_2024.TEST_TEMP[28] := B#16#0;
   S705_BT_CODE_2024.TEST_TEMP[29] := B#16#0;
   S705_BT_CODE_2024.TEST_TEMP[30] := B#16#0;
   S705_BT_CODE_2024.TEST_TEMP[31] := B#16#0;
   S705_BT_CODE_2024.TEST_TEMP[32] := B#16#0;
   S705_BT_CODE_2024.TEST_TEMP[33] := B#16#0;
   S705_BT_CODE_2024.TEST_TEMP[34] := B#16#0;
   S705_BT_CODE_2024.TEST_TEMP[35] := B#16#0;
   S705_BT_CODE_2024.TEST_TEMP[36] := B#16#0;
